LIN {X 0,Y 171.354,Z 701.949,A -85,B 0,C 180,E1 7628.432,E2 7628.432} C_VEL
LIN {X 0,Y 180.536,Z 691.15,A -85,B 0,C 180,E1 7622.276,E2 7622.276} C_VEL
LIN {X 0,Y 190.224,Z 679.335,A -85,B 0,C 180,E1 7617.222,E2 7617.222} C_VEL
LIN {X 0,Y 200.427,Z 666.059,A -85,B 0,C 180,E1 7612.87,E2 7612.87} C_VEL
LIN {X 0,Y 210.868,Z 651.279,A -85,B 0,C 180,E1 7609.131,E2 7609.131} C_VEL
LIN {X 0,Y 221.307,Z 634.876,A -85,B 0,C 180,E1 7605.912,E2 7605.912} C_VEL
LIN {X 0,Y 231.183,Z 617.293,A -85,B 0,C 180,E1 7603.218,E2 7603.218} C_VEL
LIN {X 0,Y 240.325,Z 598.504,A -85,B 0,C 180,E1 7600.964,E2 7600.964} C_VEL
LIN {X 0,Y 248.227,Z 579.366,A -85,B 0,C 180,E1 7599.16,E2 7599.16} C_VEL
LIN {X 0,Y 255.118,Z 559.071,A -85,B 0,C 180,E1 7597.658,E2 7597.658} C_VEL
LIN {X 0,Y 260.735,Z 538.067,A -85,B 0,C 180,E1 7596.463,E2 7596.463} C_VEL
LIN {X 0,Y 268.642,Z 500.013,A -85,B 0,C 180,E1 7594.871,E2 7594.871} C_VEL
LIN {X 0,Y 278.866,Z 448.019,A -85,B 0,C 180,E1 7593.295,E2 7593.295} C_VEL
LIN {X 0,Y 287.897,Z 394.54,A -85,B 0,C 180,E1 7591.964,E2 7591.964} C_VEL
LIN {X 0,Y 288.757,Z 388.485,A -85,B 0,C 180,E1 7591.797,E2 7591.797} C_VEL
LIN {X 0,Y 284.444,Z 383.003,A -85,B 0,C 180,E1 7588.674,E2 7588.674} C_VEL
LIN {X 0,Y 280.996,Z 379.022,A -85,B 0,C 180,E1 7585.729,E2 7585.729} C_VEL
LIN {X 0,Y 276.103,Z 374.241,A -85,B 0,C 180,E1 7580.344,E2 7580.344} C_VEL
LIN {X 0,Y 273.477,Z 373.45,A -85,B 0,C 180,E1 7576.133,E2 7576.133} C_VEL
LIN {X 0,Y 271.437,Z 376.229,A -85,B 0,C 180,E1 7569.97,E2 7569.97} C_VEL
LIN {X 0,Y 271.324,Z 379.346,A -85,B 0,C 180,E1 7566.56,E2 7566.56} C_VEL
LIN {X 0,Y 271.923,Z 384.024,A -85,B 0,C 180,E1 7563.057,E2 7563.057} C_VEL
LIN {X 0,Y 273.747,Z 392.011,A -85,B 0,C 180,E1 7558.64,E2 7558.64} C_VEL
LIN {X 0,Y 274.886,Z 396.29,A -85,B 0,C 180,E1 7556.725,E2 7556.725} C_VEL
LIN {X 0,Y 275.274,Z 398.796,A -85,B 0,C 180,E1 7555.994,E2 7555.994} C_VEL
LIN {X 0,Y 275.387,Z 403.134,A -85,B 0,C 180,E1 7555.297,E2 7555.297} C_VEL
LIN {X 0,Y 275.024,Z 410.299,A -85,B 0,C 180,E1 7554.636,E2 7554.636} C_VEL
LIN {X 0,Y 273.575,Z 426.263,A -85,B 0,C 180,E1 7553.562,E2 7553.562} C_VEL
LIN {X 0,Y 273.448,Z 428.423,A -85,B 0,C 180,E1 7553.346,E2 7553.346} C_VEL
LIN {X 0,Y 272.402,Z 456.029,A -85,B 0,C 180,E1 7550.133,E2 7550.133} C_VEL
LIN {X 0,Y 272.268,Z 480.855,A -85,B 0,C 180,E1 7546.766,E2 7546.766} C_VEL
LIN {X 0,Y 272.455,Z 492.691,A -85,B 0,C 180,E1 7545.052,E2 7545.052} C_VEL
LIN {X 0,Y 265.485,Z 519.701,A -85,B 0,C 180,E1 7544.247,E2 7544.247} C_VEL
LIN {X 0,Y 255.03,Z 554.502,A -85,B 0,C 180,E1 7542.869,E2 7542.869} C_VEL
LIN {X 0,Y 244.48,Z 585.093,A -85,B 0,C 180,E1 7541.222,E2 7541.222} C_VEL
LIN {X 0,Y 236.563,Z 605.451,A -85,B 0,C 180,E1 7539.768,E2 7539.768} C_VEL
LIN {X 0,Y 227.635,Z 624.889,A -85,B 0,C 180,E1 7537.94,E2 7537.94} C_VEL
LIN {X 0,Y 218.204,Z 642.726,A -85,B 0,C 180,E1 7535.763,E2 7535.763} C_VEL
LIN {X 0,Y 208.39,Z 659.271,A -85,B 0,C 180,E1 7533.18,E2 7533.18} C_VEL
LIN {X 0,Y 198.054,Z 675.047,A -85,B 0,C 180,E1 7530.015,E2 7530.015} C_VEL
LIN {X 0,Y 187.626,Z 689.669,A -85,B 0,C 180,E1 7526.234,E2 7526.234} C_VEL
LIN {X 0,Y 177.269,Z 703.298,A -85,B 0,C 180,E1 7521.628,E2 7521.628} C_VEL
LIN {X 0,Y 167.612,Z 715.397,A -85,B 0,C 180,E1 7516.203,E2 7516.203} C_VEL
LIN {X 0,Y 159.1,Z 726.025,A -85,B 0,C 180,E1 7509.867,E2 7509.867} C_VEL
LIN {X 0,Y 152.219,Z 735.127,A -85,B 0,C 180,E1 7502.589,E2 7502.589} C_VEL
LIN {X 0,Y 147.567,Z 742.333,A -85,B 0,C 180,E1 7494.782,E2 7494.782} C_VEL
LIN {X 0,Y 145.172,Z 747.597,A -85,B 0,C 180,E1 7486.798,E2 7486.798} C_VEL
LIN {X 0,Y 144.601,Z 751.03,A -85,B 0,C 180,E1 7479.15,E2 7479.15} C_VEL
LIN {X 0,Y 144.814,Z 752.641,A -85,B 0,C 180,E1 7473.166,E2 7473.166} C_VEL
LIN {X 0,Y 144.816,Z 753.275,A -85,B 0,C 180,E1 7468.021,E2 7468.021} C_VEL
LIN {X 0,Y 144.519,Z 753.042,A -85,B 0,C 180,E1 7462.046,E2 7462.046} C_VEL
LIN {X 0,Y 144.929,Z 751.416,A -85,B 0,C 180,E1 7453.98,E2 7453.98} C_VEL
LIN {X 0,Y 147.594,Z 747.947,A -85,B 0,C 180,E1 7445.164,E2 7445.164} C_VEL
LIN {X 0,Y 153.035,Z 742.69,A -85,B 0,C 180,E1 7436.713,E2 7436.713} C_VEL
LIN {X 0,Y 161.282,Z 735.568,A -85,B 0,C 180,E1 7428.917,E2 7428.917} C_VEL
LIN {X 0,Y 172.223,Z 726.333,A -85,B 0,C 180,E1 7421.884,E2 7421.884} C_VEL
LIN {X 0,Y 185.117,Z 715.226,A -85,B 0,C 180,E1 7415.885,E2 7415.885} C_VEL
LIN {X 0,Y 189.553,Z 711.162,A -85,B 0,C 180,E1 7414.101,E2 7414.101} C_VEL
LIN {X 0,Y 177.044,Z 711.814,A -85,B 0,C 180,E1 7408.687,E2 7408.687} C_VEL
LIN {X 0,Y 164.866,Z 711.841,A -85,B 0,C 180,E1 7400.222,E2 7400.222} C_VEL
LIN {X 0,Y 156.934,Z 710.739,A -85,B 0,C 180,E1 7385.85,E2 7385.85} C_VEL
LIN {X 0,Y 167.659,Z 708.493,A -85,B 0,C 180,E1 7362.65,E2 7362.65} C_VEL
LIN {X 0,Y 180.213,Z 707.275,A -85,B 0,C 180,E1 7354.299,E2 7354.299} C_VEL
LIN {X 0,Y 168.721,Z 715.346,A -85,B 0,C 180,E1 7347.935,E2 7347.935} C_VEL
LIN {X 0,Y 159.559,Z 721.376,A -85,B 0,C 180,E1 7340.991,E2 7340.991} C_VEL
LIN {X 0,Y 152.377,Z 725.891,A -85,B 0,C 180,E1 7333.034,E2 7333.034} C_VEL
LIN {X 0,Y 147.772,Z 728.661,A -85,B 0,C 180,E1 7324.637,E2 7324.637} C_VEL
LIN {X 0,Y 145.581,Z 729.803,A -85,B 0,C 180,E1 7316.515,E2 7316.515} C_VEL
LIN {X 0,Y 144.885,Z 729.625,A -85,B 0,C 180,E1 7309.345,E2 7309.345} C_VEL
LIN {X 0,Y 144.897,Z 728.45,A -85,B 0,C 180,E1 7302.353,E2 7302.353} C_VEL
LIN {X 0,Y 145.734,Z 726.021,A -85,B 0,C 180,E1 7294.723,E2 7294.723} C_VEL
LIN {X 0,Y 148.261,Z 721.791,A -85,B 0,C 180,E1 7286.491,E2 7286.491} C_VEL
LIN {X 0,Y 152.759,Z 715.974,A -85,B 0,C 180,E1 7278.676,E2 7278.676} C_VEL
LIN {X 0,Y 158.986,Z 708.791,A -85,B 0,C 180,E1 7271.673,E2 7271.673} C_VEL
LIN {X 0,Y 167.002,Z 699.89,A -85,B 0,C 180,E1 7265.223,E2 7265.223} C_VEL
LIN {X 0,Y 176.613,Z 689.064,A -85,B 0,C 180,E1 7259.369,E2 7259.369} C_VEL
LIN {X 0,Y 187.046,Z 676.723,A -85,B 0,C 180,E1 7254.363,E2 7254.363} C_VEL
LIN {X 0,Y 197.931,Z 662.854,A -85,B 0,C 180,E1 7250.093,E2 7250.093} C_VEL
LIN {X 0,Y 208.956,Z 647.38,A -85,B 0,C 180,E1 7246.446,E2 7246.446} C_VEL
LIN {X 0,Y 219.545,Z 630.725,A -85,B 0,C 180,E1 7243.415,E2 7243.415} C_VEL
LIN {X 0,Y 229.485,Z 612.921,A -85,B 0,C 180,E1 7240.893,E2 7240.893} C_VEL
LIN {X 0,Y 238.591,Z 593.934,A -85,B 0,C 180,E1 7238.789,E2 7238.789} C_VEL
LIN {X 0,Y 246.367,Z 574.632,A -85,B 0,C 180,E1 7237.111,E2 7237.111} C_VEL
LIN {X 0,Y 253.084,Z 554.191,A -85,B 0,C 180,E1 7235.721,E2 7235.721} C_VEL
LIN {X 0,Y 258.439,Z 533.188,A -85,B 0,C 180,E1 7234.629,E2 7234.629} C_VEL
LIN {X 0,Y 267.711,Z 489.4,A -85,B 0,C 180,E1 7232.935,E2 7232.935} C_VEL
LIN {X 0,Y 278.293,Z 435.561,A -85,B 0,C 180,E1 7231.428,E2 7231.428} C_VEL
LIN {X 0,Y 285.226,Z 394.061,A -85,B 0,C 180,E1 7230.419,E2 7230.419} C_VEL
LIN {X 0,Y 282.138,Z 390.149,A -85,B 0,C 180,E1 7228.018,E2 7228.018} C_VEL
LIN {X 0,Y 279.285,Z 386.715,A -85,B 0,C 180,E1 7225.443,E2 7225.443} C_VEL
LIN {X 0,Y 274.726,Z 382.112,A -85,B 0,C 180,E1 7220.228,E2 7220.228} C_VEL
LIN {X 0,Y 272.265,Z 381.361,A -85,B 0,C 180,E1 7216.207,E2 7216.207} C_VEL
LIN {X 0,Y 270.259,Z 384.053,A -85,B 0,C 180,E1 7210.23,E2 7210.23} C_VEL
LIN {X 0,Y 270.076,Z 387.081,A -85,B 0,C 180,E1 7206.911,E2 7206.911} C_VEL
LIN {X 0,Y 270.572,Z 391.825,A -85,B 0,C 180,E1 7203.39,E2 7203.39} C_VEL
LIN {X 0,Y 272.158,Z 399.486,A -85,B 0,C 180,E1 7199.159,E2 7199.159} C_VEL
LIN {X 0,Y 274.034,Z 407.176,A -85,B 0,C 180,E1 7195.921,E2 7195.921} C_VEL
LIN {X 0,Y 274.431,Z 409.099,A -85,B 0,C 180,E1 7195.299,E2 7195.299} C_VEL
LIN {X 0,Y 273.448,Z 428.423,A -85,B 0,C 180,E1 7193.346,E2 7193.346} C_VEL
LIN {X 0,Y 272.835,Z 435.664,A -85,B 0,C 180,E1 7192.766,E2 7192.766} C_VEL
LIN {X 0,Y 269.949,Z 455.079,A -85,B 0,C 180,E1 7191.849,E2 7191.849} C_VEL
LIN {X 0,Y 269.308,Z 462.105,A -85,B 0,C 180,E1 7191.184,E2 7191.184} C_VEL
LIN {X 0,Y 268.716,Z 487.169,A -85,B 0,C 180,E1 7187.674,E2 7187.674} C_VEL
LIN {X 0,Y 268.656,Z 494.996,A -85,B 0,C 180,E1 7186.554,E2 7186.554} C_VEL
LIN {X 0,Y 261.061,Z 523.455,A -85,B 0,C 180,E1 7185.692,E2 7185.692} C_VEL
LIN {X 0,Y 251.381,Z 554.96,A -85,B 0,C 180,E1 7184.477,E2 7184.477} C_VEL
LIN {X 0,Y 240.328,Z 586.648,A -85,B 0,C 180,E1 7182.82,E2 7182.82} C_VEL
LIN {X 0,Y 232.121,Z 606.804,A -85,B 0,C 180,E1 7181.377,E2 7181.377} C_VEL
LIN {X 0,Y 222.982,Z 625.913,A -85,B 0,C 180,E1 7179.58,E2 7179.58} C_VEL
LIN {X 0,Y 213.041,Z 644.023,A -85,B 0,C 180,E1 7177.367,E2 7177.367} C_VEL
LIN {X 0,Y 202.454,Z 661.114,A -85,B 0,C 180,E1 7174.659,E2 7174.659} C_VEL
LIN {X 0,Y 191.415,Z 677.098,A -85,B 0,C 180,E1 7171.347,E2 7171.347} C_VEL
LIN {X 0,Y 180.41,Z 691.618,A -85,B 0,C 180,E1 7167.395,E2 7167.395} C_VEL
LIN {X 0,Y 169.71,Z 704.845,A -85,B 0,C 180,E1 7162.641,E2 7162.641} C_VEL
LIN {X 0,Y 159.702,Z 716.716,A -85,B 0,C 180,E1 7156.968,E2 7156.968} C_VEL
LIN {X 0,Y 151.072,Z 726.931,A -85,B 0,C 180,E1 7150.436,E2 7150.436} C_VEL
LIN {X 0,Y 144.036,Z 735.711,A -85,B 0,C 180,E1 7142.782,E2 7142.782} C_VEL
LIN {X 0,Y 139.377,Z 742.546,A -85,B 0,C 180,E1 7134.587,E2 7134.587} C_VEL
LIN {X 0,Y 137.058,Z 747.585,A -85,B 0,C 180,E1 7126.093,E2 7126.093} C_VEL
LIN {X 0,Y 136.647,Z 750.774,A -85,B 0,C 180,E1 7117.991,E2 7117.991} C_VEL
LIN {X 0,Y 136.885,Z 752.225,A -85,B 0,C 180,E1 7111.674,E2 7111.674} C_VEL
LIN {X 0,Y 136.759,Z 752.604,A -85,B 0,C 180,E1 7106.227,E2 7106.227} C_VEL
LIN {X 0,Y 136.505,Z 752.171,A -85,B 0,C 180,E1 7099.448,E2 7099.448} C_VEL
LIN {X 0,Y 137.628,Z 750.098,A -85,B 0,C 180,E1 7090.476,E2 7090.476} C_VEL
LIN {X 0,Y 141.567,Z 746.099,A -85,B 0,C 180,E1 7081.136,E2 7081.136} C_VEL
LIN {X 0,Y 148.697,Z 740.161,A -85,B 0,C 180,E1 7072.272,E2 7072.272} C_VEL
LIN {X 0,Y 159.02,Z 732.136,A -85,B 0,C 180,E1 7064.209,E2 7064.209} C_VEL
LIN {X 0,Y 171.416,Z 722.422,A -85,B 0,C 180,E1 7057.506,E2 7057.506} C_VEL
LIN {X 0,Y 179.894,Z 715.408,A -85,B 0,C 180,E1 7053.869,E2 7053.869} C_VEL
LIN {X 0,Y 165.312,Z 715.757,A -85,B 0,C 180,E1 7046.587,E2 7046.587} C_VEL
LIN {X 0,Y 154.531,Z 715.3,A -85,B 0,C 180,E1 7036.926,E2 7036.926} C_VEL
LIN {X 0,Y 149.737,Z 714.176,A -85,B 0,C 180,E1 7024.979,E2 7024.979} C_VEL
LIN {X 0,Y 160.695,Z 711.869,A -85,B 0,C 180,E1 7001.873,E2 7001.873} C_VEL
LIN {X 0,Y 171.293,Z 710.841,A -85,B 0,C 180,E1 6994.53,E2 6994.53} C_VEL
LIN {X 0,Y 159.716,Z 718.272,A -85,B 0,C 180,E1 6987.85,E2 6987.85} C_VEL
LIN {X 0,Y 150.382,Z 723.839,A -85,B 0,C 180,E1 6980.334,E2 6980.334} C_VEL
LIN {X 0,Y 143.279,Z 727.812,A -85,B 0,C 180,E1 6971.693,E2 6971.693} C_VEL
LIN {X 0,Y 139.036,Z 730,A -85,B 0,C 180,E1 6962.641,E2 6962.641} C_VEL
LIN {X 0,Y 137.309,Z 730.53,A -85,B 0,C 180,E1 6954.46,E2 6954.46} C_VEL
LIN {X 0,Y 136.849,Z 729.926,A -85,B 0,C 180,E1 6946.833,E2 6946.833} C_VEL
LIN {X 0,Y 137.087,Z 728.42,A -85,B 0,C 180,E1 6939.658,E2 6939.658} C_VEL
LIN {X 0,Y 138.427,Z 725.493,A -85,B 0,C 180,E1 6931.656,E2 6931.656} C_VEL
LIN {X 0,Y 141.776,Z 720.799,A -85,B 0,C 180,E1 6923.115,E2 6923.115} C_VEL
LIN {X 0,Y 147.636,Z 714.09,A -85,B 0,C 180,E1 6914.686,E2 6914.686} C_VEL
LIN {X 0,Y 155.429,Z 705.841,A -85,B 0,C 180,E1 6907.296,E2 6907.296} C_VEL
LIN {X 0,Y 165.159,Z 695.6,A -85,B 0,C 180,E1 6900.636,E2 6900.636} C_VEL
LIN {X 0,Y 175.99,Z 683.736,A -85,B 0,C 180,E1 6894.984,E2 6894.984} C_VEL
LIN {X 0,Y 187.476,Z 670.238,A -85,B 0,C 180,E1 6890.209,E2 6890.209} C_VEL
LIN {X 0,Y 198.57,Z 655.944,A -85,B 0,C 180,E1 6886.383,E2 6886.383} C_VEL
LIN {X 0,Y 209.615,Z 640.112,A -85,B 0,C 180,E1 6883.13,E2 6883.13} C_VEL
LIN {X 0,Y 220.041,Z 623.212,A -85,B 0,C 180,E1 6880.438,E2 6880.438} C_VEL
LIN {X 0,Y 229.654,Z 605.283,A -85,B 0,C 180,E1 6878.201,E2 6878.201} C_VEL
LIN {X 0,Y 238.329,Z 586.285,A -85,B 0,C 180,E1 6876.342,E2 6876.342} C_VEL
LIN {X 0,Y 245.568,Z 567.229,A -85,B 0,C 180,E1 6874.872,E2 6874.872} C_VEL
LIN {X 0,Y 251.885,Z 546.585,A -85,B 0,C 180,E1 6873.633,E2 6873.633} C_VEL
LIN {X 0,Y 258.787,Z 517.082,A -85,B 0,C 180,E1 6872.31,E2 6872.31} C_VEL
LIN {X 0,Y 267.881,Z 474.899,A -85,B 0,C 180,E1 6870.894,E2 6870.894} C_VEL
LIN {X 0,Y 278.004,Z 422.549,A -85,B 0,C 180,E1 6869.551,E2 6869.551} C_VEL
LIN {X 0,Y 281.82,Z 399.7,A -85,B 0,C 180,E1 6869.01,E2 6869.01} C_VEL
LIN {X 0,Y 277.532,Z 394.401,A -85,B 0,C 180,E1 6865.159,E2 6865.159} C_VEL
LIN {X 0,Y 273.269,Z 389.97,A -85,B 0,C 180,E1 6860.118,E2 6860.118} C_VEL
LIN {X 0,Y 271.014,Z 389.266,A -85,B 0,C 180,E1 6856.284,E2 6856.284} C_VEL
LIN {X 0,Y 268.974,Z 392.056,A -85,B 0,C 180,E1 6850.279,E2 6850.279} C_VEL
LIN {X 0,Y 268.78,Z 394.936,A -85,B 0,C 180,E1 6847.16,E2 6847.16} C_VEL
LIN {X 0,Y 269.175,Z 399.61,A -85,B 0,C 180,E1 6843.728,E2 6843.728} C_VEL
LIN {X 0,Y 270.526,Z 406.946,A -85,B 0,C 180,E1 6839.683,E2 6839.683} C_VEL
LIN {X 0,Y 272.103,Z 414.302,A -85,B 0,C 180,E1 6836.577,E2 6836.577} C_VEL
LIN {X 0,Y 270.3,Z 442.419,A -85,B 0,C 180,E1 6833.589,E2 6833.589} C_VEL
LIN {X 0,Y 269.308,Z 462.105,A -85,B 0,C 180,E1 6831.184,E2 6831.184} C_VEL
LIN {X 0,Y 268.709,Z 469.106,A -85,B 0,C 180,E1 6830.479,E2 6830.479} C_VEL
LIN {X 0,Y 265.764,Z 488.052,A -85,B 0,C 180,E1 6829.195,E2 6829.195} C_VEL
LIN {X 0,Y 265.158,Z 494.824,A -85,B 0,C 180,E1 6828.404,E2 6828.404} C_VEL
LIN {X 0,Y 264.979,Z 497.272,A -85,B 0,C 180,E1 6828.09,E2 6828.09} C_VEL
LIN {X 0,Y 256.396,Z 528.682,A -85,B 0,C 180,E1 6827.139,E2 6827.139} C_VEL
LIN {X 0,Y 245.452,Z 562.722,A -85,B 0,C 180,E1 6825.812,E2 6825.812} C_VEL
LIN {X 0,Y 235.247,Z 590.673,A -85,B 0,C 180,E1 6824.297,E2 6824.297} C_VEL
LIN {X 0,Y 227.439,Z 608.962,A -85,B 0,C 180,E1 6822.972,E2 6822.972} C_VEL
LIN {X 0,Y 217.978,Z 628.013,A -85,B 0,C 180,E1 6821.177,E2 6821.177} C_VEL
LIN {X 0,Y 207.383,Z 646.391,A -85,B 0,C 180,E1 6818.895,E2 6818.895} C_VEL
LIN {X 0,Y 196.267,Z 663.341,A -85,B 0,C 180,E1 6816.126,E2 6816.126} C_VEL
LIN {X 0,Y 184.568,Z 679.376,A -85,B 0,C 180,E1 6812.677,E2 6812.677} C_VEL
LIN {X 0,Y 173.275,Z 693.522,A -85,B 0,C 180,E1 6808.65,E2 6808.65} C_VEL
LIN {X 0,Y 162.092,Z 706.598,A -85,B 0,C 180,E1 6803.69,E2 6803.69} C_VEL
LIN {X 0,Y 151.554,Z 718.304,A -85,B 0,C 180,E1 6797.637,E2 6797.637} C_VEL
LIN {X 0,Y 142.644,Z 728.178,A -85,B 0,C 180,E1 6790.683,E2 6790.683} C_VEL
LIN {X 0,Y 135.559,Z 736.567,A -85,B 0,C 180,E1 6782.576,E2 6782.576} C_VEL
LIN {X 0,Y 130.99,Z 743.072,A -85,B 0,C 180,E1 6773.862,E2 6773.862} C_VEL
LIN {X 0,Y 128.899,Z 747.786,A -85,B 0,C 180,E1 6764.831,E2 6764.831} C_VEL
LIN {X 0,Y 128.716,Z 750.513,A -85,B 0,C 180,E1 6756.691,E2 6756.691} C_VEL
LIN {X 0,Y 128.939,Z 751.655,A -85,B 0,C 180,E1 6750.444,E2 6750.444} C_VEL
LIN {X 0,Y 128.695,Z 751.92,A -85,B 0,C 180,E1 6744.65,E2 6744.65} C_VEL
LIN {X 0,Y 128.67,Z 751.118,A -85,B 0,C 180,E1 6736.244,E2 6736.244} C_VEL
LIN {X 0,Y 130.795,Z 748.594,A -85,B 0,C 180,E1 6726.536,E2 6726.536} C_VEL
LIN {X 0,Y 136.327,Z 744.053,A -85,B 0,C 180,E1 6716.627,E2 6716.627} C_VEL
LIN {X 0,Y 145.281,Z 737.569,A -85,B 0,C 180,E1 6707.587,E2 6707.587} C_VEL
LIN {X 0,Y 156.702,Z 729.392,A -85,B 0,C 180,E1 6700.032,E2 6700.032} C_VEL
LIN {X 0,Y 170.19,Z 719.296,A -85,B 0,C 180,E1 6693.621,E2 6693.621} C_VEL
LIN {X 0,Y 154.36,Z 719.231,A -85,B 0,C 180,E1 6684.49,E2 6684.49} C_VEL
LIN {X 0,Y 143.397,Z 718.1,A -85,B 0,C 180,E1 6670.038,E2 6670.038} C_VEL
LIN {X 0,Y 154.109,Z 715.004,A -85,B 0,C 180,E1 6640.676,E2 6640.676} C_VEL
LIN {X 0,Y 162.224,Z 714.235,A -85,B 0,C 180,E1 6634.733,E2 6634.733} C_VEL
LIN {X 0,Y 150.963,Z 720.78,A -85,B 0,C 180,E1 6627.971,E2 6627.971} C_VEL
LIN {X 0,Y 141.536,Z 725.832,A -85,B 0,C 180,E1 6619.993,E2 6619.993} C_VEL
LIN {X 0,Y 134.84,Z 729.141,A -85,B 0,C 180,E1 6611.297,E2 6611.297} C_VEL
LIN {X 0,Y 130.765,Z 730.897,A -85,B 0,C 180,E1 6601.844,E2 6601.844} C_VEL
LIN {X 0,Y 129.159,Z 731.134,A -85,B 0,C 180,E1 6592.892,E2 6592.892} C_VEL
LIN {X 0,Y 128.875,Z 730.299,A -85,B 0,C 180,E1 6585.296,E2 6585.296} C_VEL
LIN {X 0,Y 129.368,Z 728.333,A -85,B 0,C 180,E1 6577.104,E2 6577.104} C_VEL
LIN {X 0,Y 131.435,Z 724.876,A -85,B 0,C 180,E1 6568.257,E2 6568.257} C_VEL
LIN {X 0,Y 135.782,Z 719.681,A -85,B 0,C 180,E1 6559.392,E2 6559.392} C_VEL
LIN {X 0,Y 142.46,Z 712.772,A -85,B 0,C 180,E1 6551.165,E2 6551.165} C_VEL
LIN {X 0,Y 151.325,Z 704.001,A -85,B 0,C 180,E1 6543.725,E2 6543.725} C_VEL
LIN {X 0,Y 161.537,Z 693.741,A -85,B 0,C 180,E1 6537.419,E2 6537.419} C_VEL
LIN {X 0,Y 172.62,Z 682.015,A -85,B 0,C 180,E1 6532.123,E2 6532.123} C_VEL
LIN {X 0,Y 184.126,Z 668.837,A -85,B 0,C 180,E1 6527.674,E2 6527.674} C_VEL
LIN {X 0,Y 195.756,Z 654.155,A -85,B 0,C 180,E1 6523.931,E2 6523.931} C_VEL
LIN {X 0,Y 207.256,Z 637.837,A -85,B 0,C 180,E1 6520.764,E2 6520.764} C_VEL
LIN {X 0,Y 218.052,Z 620.358,A -85,B 0,C 180,E1 6518.15,E2 6518.15} C_VEL
LIN {X 0,Y 227.942,Z 601.777,A -85,B 0,C 180,E1 6515.994,E2 6515.994} C_VEL
LIN {X 0,Y 236.523,Z 582.728,A -85,B 0,C 180,E1 6514.265,E2 6514.265} C_VEL
LIN {X 0,Y 243.955,Z 562.676,A -85,B 0,C 180,E1 6512.839,E2 6512.839} C_VEL
LIN {X 0,Y 250.174,Z 541.384,A -85,B 0,C 180,E1 6511.676,E2 6511.676} C_VEL
LIN {X 0,Y 259.603,Z 500.631,A -85,B 0,C 180,E1 6510.042,E2 6510.042} C_VEL
LIN {X 0,Y 269.641,Z 454.025,A -85,B 0,C 180,E1 6508.722,E2 6508.722} C_VEL
LIN {X 0,Y 278.539,Z 405.648,A -85,B 0,C 180,E1 6507.586,E2 6507.586} C_VEL
LIN {X 0,Y 275.56,Z 401.887,A -85,B 0,C 180,E1 6504.663,E2 6504.663} C_VEL
LIN {X 0,Y 271.804,Z 397.826,A -85,B 0,C 180,E1 6500.006,E2 6500.006} C_VEL
LIN {X 0,Y 269.673,Z 397.154,A -85,B 0,C 180,E1 6496.367,E2 6496.367} C_VEL
LIN {X 0,Y 267.682,Z 399.855,A -85,B 0,C 180,E1 6490.547,E2 6490.547} C_VEL
LIN {X 0,Y 267.443,Z 402.648,A -85,B 0,C 180,E1 6487.519,E2 6487.519} C_VEL
LIN {X 0,Y 267.718,Z 407.375,A -85,B 0,C 180,E1 6484.07,E2 6484.07} C_VEL
LIN {X 0,Y 268.86,Z 414.392,A -85,B 0,C 180,E1 6480.214,E2 6480.214} C_VEL
LIN {X 0,Y 269.859,Z 420.094,A -85,B 0,C 180,E1 6477.798,E2 6477.798} C_VEL
LIN {X 0,Y 267.706,Z 446.388,A -85,B 0,C 180,E1 6474.965,E2 6474.965} C_VEL
LIN {X 0,Y 266.016,Z 471.924,A -85,B 0,C 180,E1 6471.748,E2 6471.748} C_VEL
LIN {X 0,Y 265.158,Z 494.824,A -85,B 0,C 180,E1 6468.404,E2 6468.404} C_VEL
LIN {X 0,Y 264.609,Z 498.077,A -85,B 0,C 180,E1 6468.164,E2 6468.164} C_VEL
LIN {X 0,Y 263.21,Z 502.217,A -85,B 0,C 180,E1 6468.258,E2 6468.258} C_VEL
LIN {X 0,Y 258.133,Z 513.262,A -85,B 0,C 180,E1 6469.155,E2 6469.155} C_VEL
LIN {X 0,Y 256.778,Z 517.033,A -85,B 0,C 180,E1 6469.182,E2 6469.182} C_VEL
LIN {X 0,Y 246.767,Z 549.705,A -85,B 0,C 180,E1 6468.075,E2 6468.075} C_VEL
LIN {X 0,Y 235.377,Z 582.079,A -85,B 0,C 180,E1 6466.598,E2 6466.598} C_VEL
LIN {X 0,Y 226.9,Z 602.616,A -85,B 0,C 180,E1 6465.295,E2 6465.295} C_VEL
LIN {X 0,Y 217.706,Z 621.428,A -85,B 0,C 180,E1 6463.713,E2 6463.713} C_VEL
LIN {X 0,Y 207.444,Z 639.576,A -85,B 0,C 180,E1 6461.716,E2 6461.716} C_VEL
LIN {X 0,Y 196.658,Z 656.347,A -85,B 0,C 180,E1 6459.309,E2 6459.309} C_VEL
LIN {X 0,Y 185.1,Z 672.382,A -85,B 0,C 180,E1 6456.289,E2 6456.289} C_VEL
LIN {X 0,Y 173.381,Z 687.06,A -85,B 0,C 180,E1 6452.633,E2 6452.633} C_VEL
LIN {X 0,Y 161.435,Z 700.69,A -85,B 0,C 180,E1 6448.05,E2 6448.05} C_VEL
LIN {X 0,Y 150.046,Z 712.887,A -85,B 0,C 180,E1 6442.464,E2 6442.464} C_VEL
LIN {X 0,Y 139.708,Z 723.626,A -85,B 0,C 180,E1 6435.698,E2 6435.698} C_VEL
LIN {X 0,Y 131.417,Z 732.411,A -85,B 0,C 180,E1 6428.044,E2 6428.044} C_VEL
LIN {X 0,Y 125.206,Z 739.756,A -85,B 0,C 180,E1 6419.151,E2 6419.151} C_VEL
LIN {X 0,Y 121.7,Z 745.246,A -85,B 0,C 180,E1 6409.684,E2 6409.684} C_VEL
LIN {X 0,Y 120.666,Z 748.836,A -85,B 0,C 180,E1 6400.503,E2 6400.503} C_VEL
LIN {X 0,Y 120.892,Z 750.527,A -85,B 0,C 180,E1 6393.318,E2 6393.318} C_VEL
LIN {X 0,Y 120.884,Z 751.184,A -85,B 0,C 180,E1 6387.629,E2 6387.629} C_VEL
LIN {X 0,Y 120.547,Z 751.088,A -85,B 0,C 180,E1 6380.45,E2 6380.45} C_VEL
LIN {X 0,Y 121.482,Z 749.628,A -85,B 0,C 180,E1 6370.778,E2 6370.778} C_VEL
LIN {X 0,Y 125.495,Z 746.319,A -85,B 0,C 180,E1 6360.397,E2 6360.397} C_VEL
LIN {X 0,Y 133.3,Z 741.012,A -85,B 0,C 180,E1 6350.388,E2 6350.388} C_VEL
LIN {X 0,Y 143.943,Z 734.076,A -85,B 0,C 180,E1 6341.99,E2 6341.99} C_VEL
LIN {X 0,Y 157.18,Z 725.207,A -85,B 0,C 180,E1 6334.854,E2 6334.854} C_VEL
LIN {X 0,Y 160.523,Z 722.807,A -85,B 0,C 180,E1 6333.334,E2 6333.334} C_VEL
LIN {X 0,Y 145.642,Z 722.467,A -85,B 0,C 180,E1 6323.893,E2 6323.893} C_VEL
LIN {X 0,Y 135.208,Z 720.885,A -85,B 0,C 180,E1 6306.367,E2 6306.367} C_VEL
LIN {X 0,Y 149.221,Z 717.769,A -85,B 0,C 180,E1 6277.96,E2 6277.96} C_VEL
LIN {X 0,Y 153.292,Z 717.333,A -85,B 0,C 180,E1 6275.046,E2 6275.046} C_VEL
LIN {X 0,Y 141.241,Z 723.643,A -85,B 0,C 180,E1 6267.397,E2 6267.397} C_VEL
LIN {X 0,Y 131.452,Z 728.258,A -85,B 0,C 180,E1 6258.196,E2 6258.196} C_VEL
LIN {X 0,Y 125.188,Z 730.881,A -85,B 0,C 180,E1 6248.488,E2 6248.488} C_VEL
LIN {X 0,Y 121.937,Z 731.86,A -85,B 0,C 180,E1 6238.399,E2 6238.399} C_VEL
LIN {X 0,Y 120.975,Z 731.553,A -85,B 0,C 180,E1 6229.809,E2 6229.809} C_VEL
LIN {X 0,Y 120.982,Z 730.257,A -85,B 0,C 180,E1 6221.925,E2 6221.925} C_VEL
LIN {X 0,Y 122.119,Z 727.691,A -85,B 0,C 180,E1 6212.817,E2 6212.817} C_VEL
LIN {X 0,Y 125.261,Z 723.628,A -85,B 0,C 180,E1 6203.584,E2 6203.584} C_VEL
LIN {X 0,Y 131.312,Z 717.409,A -85,B 0,C 180,E1 6194.091,E2 6194.091} C_VEL
LIN {X 0,Y 139.562,Z 709.661,A -85,B 0,C 180,E1 6185.899,E2 6185.899} C_VEL
LIN {X 0,Y 149.926,Z 699.969,A -85,B 0,C 180,E1 6178.656,E2 6178.656} C_VEL
LIN {X 0,Y 161.459,Z 688.696,A -85,B 0,C 180,E1 6172.636,E2 6172.636} C_VEL
LIN {X 0,Y 173.637,Z 675.844,A -85,B 0,C 180,E1 6167.645,E2 6167.645} C_VEL
LIN {X 0,Y 185.363,Z 662.258,A -85,B 0,C 180,E1 6163.714,E2 6163.714} C_VEL
LIN {X 0,Y 197.348,Z 646.732,A -85,B 0,C 180,E1 6160.315,E2 6160.315} C_VEL
LIN {X 0,Y 209.062,Z 629.495,A -85,B 0,C 180,E1 6157.448,E2 6157.448} C_VEL
LIN {X 0,Y 219.942,Z 610.979,A -85,B 0,C 180,E1 6155.087,E2 6155.087} C_VEL
LIN {X 0,Y 229.439,Z 591.945,A -85,B 0,C 180,E1 6153.207,E2 6153.207} C_VEL
LIN {X 0,Y 237.831,Z 571.656,A -85,B 0,C 180,E1 6151.645,E2 6151.645} C_VEL
LIN {X 0,Y 244.659,Z 551.112,A -85,B 0,C 180,E1 6150.424,E2 6150.424} C_VEL
LIN {X 0,Y 251.802,Z 523.021,A -85,B 0,C 180,E1 6149.167,E2 6149.167} C_VEL
LIN {X 0,Y 261.39,Z 481.732,A -85,B 0,C 180,E1 6147.787,E2 6147.787} C_VEL
LIN {X 0,Y 271.741,Z 431.737,A -85,B 0,C 180,E1 6146.562,E2 6146.562} C_VEL
LIN {X 0,Y 275.361,Z 411.62,A -85,B 0,C 180,E1 6146.097,E2 6146.097} C_VEL
LIN {X 0,Y 273.14,Z 408.943,A -85,B 0,C 180,E1 6143.746,E2 6143.746} C_VEL
LIN {X 0,Y 270.249,Z 405.666,A -85,B 0,C 180,E1 6139.901,E2 6139.901} C_VEL
LIN {X 0,Y 268.296,Z 405.036,A -85,B 0,C 180,E1 6136.454,E2 6136.454} C_VEL
LIN {X 0,Y 266.302,Z 407.634,A -85,B 0,C 180,E1 6130.821,E2 6130.821} C_VEL
LIN {X 0,Y 266.006,Z 410.335,A -85,B 0,C 180,E1 6127.886,E2 6127.886} C_VEL
LIN {X 0,Y 266.157,Z 415.111,A -85,B 0,C 180,E1 6124.418,E2 6124.418} C_VEL
LIN {X 0,Y 267.114,Z 421.92,A -85,B 0,C 180,E1 6120.698,E2 6120.698} C_VEL
LIN {X 0,Y 267.66,Z 425.756,A -85,B 0,C 180,E1 6119.064,E2 6119.064} C_VEL
LIN {X 0,Y 264.823,Z 454.145,A -85,B 0,C 180,E1 6115.914,E2 6115.914} C_VEL
LIN {X 0,Y 262.74,Z 480.368,A -85,B 0,C 180,E1 6112.484,E2 6112.484} C_VEL
LIN {X 0,Y 261.59,Z 499.478,A -85,B 0,C 180,E1 6109.672,E2 6109.672} C_VEL
LIN {X 0,Y 256.778,Z 517.033,A -85,B 0,C 180,E1 6109.182,E2 6109.182} C_VEL
LIN {X 0,Y 254.311,Z 524.379,A -85,B 0,C 180,E1 6109.196,E2 6109.196} C_VEL
LIN {X 0,Y 246.54,Z 542.774,A -85,B 0,C 180,E1 6109.865,E2 6109.865} C_VEL
LIN {X 0,Y 243.816,Z 550.01,A -85,B 0,C 180,E1 6109.811,E2 6109.811} C_VEL
LIN {X 0,Y 233.133,Z 580.237,A -85,B 0,C 180,E1 6108.517,E2 6108.517} C_VEL
LIN {X 0,Y 224.777,Z 600.351,A -85,B 0,C 180,E1 6107.324,E2 6107.324} C_VEL
LIN {X 0,Y 215.958,Z 618.332,A -85,B 0,C 180,E1 6105.92,E2 6105.92} C_VEL
LIN {X 0,Y 205.839,Z 636.126,A -85,B 0,C 180,E1 6104.107,E2 6104.107} C_VEL
LIN {X 0,Y 194.691,Z 653.269,A -85,B 0,C 180,E1 6101.821,E2 6101.821} C_VEL
LIN {X 0,Y 183.088,Z 669.096,A -85,B 0,C 180,E1 6099.041,E2 6099.041} C_VEL
LIN {X 0,Y 171.206,Z 683.678,A -85,B 0,C 180,E1 6095.65,E2 6095.65} C_VEL
LIN {X 0,Y 159.28,Z 697.026,A -85,B 0,C 180,E1 6091.5,E2 6091.5} C_VEL
LIN {X 0,Y 146.981,Z 709.789,A -85,B 0,C 180,E1 6086.09,E2 6086.09} C_VEL
LIN {X 0,Y 135.602,Z 720.933,A -85,B 0,C 180,E1 6079.417,E2 6079.417} C_VEL
LIN {X 0,Y 126.212,Z 730.077,A -85,B 0,C 180,E1 6071.716,E2 6071.716} C_VEL
LIN {X 0,Y 118.587,Z 738.106,A -85,B 0,C 180,E1 6062.084,E2 6062.084} C_VEL
LIN {X 0,Y 114.197,Z 743.984,A -85,B 0,C 180,E1 6051.866,E2 6051.866} C_VEL
LIN {X 0,Y 112.717,Z 747.868,A -85,B 0,C 180,E1 6041.771,E2 6041.771} C_VEL
LIN {X 0,Y 112.91,Z 749.789,A -85,B 0,C 180,E1 6033.553,E2 6033.553} C_VEL
LIN {X 0,Y 112.93,Z 750.443,A -85,B 0,C 180,E1 6027.97,E2 6027.97} C_VEL
LIN {X 0,Y 112.568,Z 750.488,A -85,B 0,C 180,E1 6020.369,E2 6020.369} C_VEL
LIN {X 0,Y 113.637,Z 749.148,A -85,B 0,C 180,E1 6009.93,E2 6009.93} C_VEL
LIN {X 0,Y 118.209,Z 745.904,A -85,B 0,C 180,E1 5998.68,E2 5998.68} C_VEL
LIN {X 0,Y 126.547,Z 740.832,A -85,B 0,C 180,E1 5988.417,E2 5988.417} C_VEL
LIN {X 0,Y 138.507,Z 733.698,A -85,B 0,C 180,E1 5979.428,E2 5979.428} C_VEL
LIN {X 0,Y 150.869,Z 726.021,A -85,B 0,C 180,E1 5973.03,E2 5973.03} C_VEL
LIN {X 0,Y 136.9,Z 725.437,A -85,B 0,C 180,E1 5963.227,E2 5963.227} C_VEL
LIN {X 0,Y 127.754,Z 723.806,A -85,B 0,C 180,E1 5946.289,E2 5946.289} C_VEL
LIN {X 0,Y 140.941,Z 720.674,A -85,B 0,C 180,E1 5917.913,E2 5917.913} C_VEL
LIN {X 0,Y 144.162,Z 720.373,A -85,B 0,C 180,E1 5915.311,E2 5915.311} C_VEL
LIN {X 0,Y 132.035,Z 726.048,A -85,B 0,C 180,E1 5907.202,E2 5907.202} C_VEL
LIN {X 0,Y 122.738,Z 729.901,A -85,B 0,C 180,E1 5897.845,E2 5897.845} C_VEL
LIN {X 0,Y 116.625,Z 732.049,A -85,B 0,C 180,E1 5887.497,E2 5887.497} C_VEL
LIN {X 0,Y 113.728,Z 732.566,A -85,B 0,C 180,E1 5877.205,E2 5877.205} C_VEL
LIN {X 0,Y 112.936,Z 731.902,A -85,B 0,C 180,E1 5868.052,E2 5868.052} C_VEL
LIN {X 0,Y 113.144,Z 730.434,A -85,B 0,C 180,E1 5859.667,E2 5859.667} C_VEL
LIN {X 0,Y 114.789,Z 727.516,A -85,B 0,C 180,E1 5850.001,E2 5850.001} C_VEL
LIN {X 0,Y 119.009,Z 722.831,A -85,B 0,C 180,E1 5839.839,E2 5839.839} C_VEL
LIN {X 0,Y 125.9,Z 716.472,A -85,B 0,C 180,E1 5830.516,E2 5830.516} C_VEL
LIN {X 0,Y 135.245,Z 708.308,A -85,B 0,C 180,E1 5822.242,E2 5822.242} C_VEL
LIN {X 0,Y 146.667,Z 698.143,A -85,B 0,C 180,E1 5815.066,E2 5815.066} C_VEL
LIN {X 0,Y 158.466,Z 686.99,A -85,B 0,C 180,E1 5809.467,E2 5809.467} C_VEL
LIN {X 0,Y 171.383,Z 673.681,A -85,B 0,C 180,E1 5804.623,E2 5804.623} C_VEL
LIN {X 0,Y 183.692,Z 659.588,A -85,B 0,C 180,E1 5800.836,E2 5800.836} C_VEL
LIN {X 0,Y 196.2,Z 643.463,A -85,B 0,C 180,E1 5797.586,E2 5797.586} C_VEL
LIN {X 0,Y 207.555,Z 626.742,A -85,B 0,C 180,E1 5795.021,E2 5795.021} C_VEL
LIN {X 0,Y 218.361,Z 608.293,A -85,B 0,C 180,E1 5792.836,E2 5792.836} C_VEL
LIN {X 0,Y 227.709,Z 589.447,A -85,B 0,C 180,E1 5791.104,E2 5791.104} C_VEL
LIN {X 0,Y 235.896,Z 569.492,A -85,B 0,C 180,E1 5789.669,E2 5789.669} C_VEL
LIN {X 0,Y 242.67,Z 548.804,A -85,B 0,C 180,E1 5788.522,E2 5788.522} C_VEL
LIN {X 0,Y 251.957,Z 512.333,A -85,B 0,C 180,E1 5787.034,E2 5787.034} C_VEL
LIN {X 0,Y 261.592,Z 471.098,A -85,B 0,C 180,E1 5785.826,E2 5785.826} C_VEL
LIN {X 0,Y 271.58,Z 422.04,A -85,B 0,C 180,E1 5784.715,E2 5784.715} C_VEL
LIN {X 0,Y 272.327,Z 417.667,A -85,B 0,C 180,E1 5784.572,E2 5784.572} C_VEL
LIN {X 0,Y 268.555,Z 413.462,A -85,B 0,C 180,E1 5779.619,E2 5779.619} C_VEL
LIN {X 0,Y 266.863,Z 412.907,A -85,B 0,C 180,E1 5776.545,E2 5776.545} C_VEL
LIN {X 0,Y 264.859,Z 415.458,A -85,B 0,C 180,E1 5771.035,E2 5771.035} C_VEL
LIN {X 0,Y 264.531,Z 418.012,A -85,B 0,C 180,E1 5768.259,E2 5768.259} C_VEL
LIN {X 0,Y 264.565,Z 422.834,A -85,B 0,C 180,E1 5764.77,E2 5764.77} C_VEL
LIN {X 0,Y 265.313,Z 429.426,A -85,B 0,C 180,E1 5761.188,E2 5761.188} C_VEL
LIN {X 0,Y 265.512,Z 431.556,A -85,B 0,C 180,E1 5760.324,E2 5760.324} C_VEL
LIN {X 0,Y 262.124,Z 460.31,A -85,B 0,C 180,E1 5757.063,E2 5757.063} C_VEL
LIN {X 0,Y 259.613,Z 486.376,A -85,B 0,C 180,E1 5753.563,E2 5753.563} C_VEL
LIN {X 0,Y 258.39,Z 501.571,A -85,B 0,C 180,E1 5751.29,E2 5751.29} C_VEL
LIN {X 0,Y 248.519,Z 535.696,A -85,B 0,C 180,E1 5750.298,E2 5750.298} C_VEL
LIN {X 0,Y 243.816,Z 550.01,A -85,B 0,C 180,E1 5749.811,E2 5749.811} C_VEL
LIN {X 0,Y 241.066,Z 557.266,A -85,B 0,C 180,E1 5749.767,E2 5749.767} C_VEL
LIN {X 0,Y 232.138,Z 576.405,A -85,B 0,C 180,E1 5750.386,E2 5750.386} C_VEL
LIN {X 0,Y 229.54,Z 582.459,A -85,B 0,C 180,E1 5750.271,E2 5750.271} C_VEL
LIN {X 0,Y 220.946,Z 602.34,A -85,B 0,C 180,E1 5749.112,E2 5749.112} C_VEL
LIN {X 0,Y 211.352,Z 621.037,A -85,B 0,C 180,E1 5747.661,E2 5747.661} C_VEL
LIN {X 0,Y 200.145,Z 639.801,A -85,B 0,C 180,E1 5745.733,E2 5745.733} C_VEL
LIN {X 0,Y 188.024,Z 657.303,A -85,B 0,C 180,E1 5743.313,E2 5743.313} C_VEL
LIN {X 0,Y 175.572,Z 673.18,A -85,B 0,C 180,E1 5740.368,E2 5740.368} C_VEL
LIN {X 0,Y 163.14,Z 687.411,A -85,B 0,C 180,E1 5736.827,E2 5736.827} C_VEL
LIN {X 0,Y 150.081,Z 700.987,A -85,B 0,C 180,E1 5732.204,E2 5732.204} C_VEL
LIN {X 0,Y 137.593,Z 713.015,A -85,B 0,C 180,E1 5726.478,E2 5726.478} C_VEL
LIN {X 0,Y 126.281,Z 723.41,A -85,B 0,C 180,E1 5719.472,E2 5719.472} C_VEL
LIN {X 0,Y 116.491,Z 732.374,A -85,B 0,C 180,E1 5710.716,E2 5710.716} C_VEL
LIN {X 0,Y 109.533,Z 739.383,A -85,B 0,C 180,E1 5700.742,E2 5700.742} C_VEL
LIN {X 0,Y 105.679,Z 744.588,A -85,B 0,C 180,E1 5689.913,E2 5689.913} C_VEL
LIN {X 0,Y 104.709,Z 747.927,A -85,B 0,C 180,E1 5679.341,E2 5679.341} C_VEL
LIN {X 0,Y 104.985,Z 749.307,A -85,B 0,C 180,E1 5672.182,E2 5672.182} C_VEL
LIN {X 0,Y 104.864,Z 749.842,A -85,B 0,C 180,E1 5666.172,E2 5666.172} C_VEL
LIN {X 0,Y 104.676,Z 749.599,A -85,B 0,C 180,E1 5656.746,E2 5656.746} C_VEL
LIN {X 0,Y 107.005,Z 747.809,A -85,B 0,C 180,E1 5645.005,E2 5645.005} C_VEL
LIN {X 0,Y 113.502,Z 744.099,A -85,B 0,C 180,E1 5633.199,E2 5633.199} C_VEL
LIN {X 0,Y 124.049,Z 738.458,A -85,B 0,C 180,E1 5622.82,E2 5622.82} C_VEL
LIN {X 0,Y 137.234,Z 731.213,A -85,B 0,C 180,E1 5614.582,E2 5614.582} C_VEL
LIN {X 0,Y 140.98,Z 728.956,A -85,B 0,C 180,E1 5612.615,E2 5612.615} C_VEL
LIN {X 0,Y 127.052,Z 728.036,A -85,B 0,C 180,E1 5601.222,E2 5601.222} C_VEL
LIN {X 0,Y 120.05,Z 725.9,A -85,B 0,C 180,E1 5579.998,E2 5579.998} C_VEL
LIN {X 0,Y 135.017,Z 723.116,A -85,B 0,C 180,E1 5555.627,E2 5555.627} C_VEL
LIN {X 0,Y 122.73,Z 728.218,A -85,B 0,C 180,E1 5546.916,E2 5546.916} C_VEL
LIN {X 0,Y 113.335,Z 731.552,A -85,B 0,C 180,E1 5536.516,E2 5536.516} C_VEL
LIN {X 0,Y 107.641,Z 733.086,A -85,B 0,C 180,E1 5525.164,E2 5525.164} C_VEL
LIN {X 0,Y 105.354,Z 733.073,A -85,B 0,C 180,E1 5514.34,E2 5514.34} C_VEL
LIN {X 0,Y 104.95,Z 732.101,A -85,B 0,C 180,E1 5504.907,E2 5504.907} C_VEL
LIN {X 0,Y 105.626,Z 730.058,A -85,B 0,C 180,E1 5495.433,E2 5495.433} C_VEL
LIN {X 0,Y 108.476,Z 726.45,A -85,B 0,C 180,E1 5484.712,E2 5484.712} C_VEL
LIN {X 0,Y 114.278,Z 721.083,A -85,B 0,C 180,E1 5474.25,E2 5474.25} C_VEL
LIN {X 0,Y 122.822,Z 714.001,A -85,B 0,C 180,E1 5464.957,E2 5464.957} C_VEL
LIN {X 0,Y 133.744,Z 705.026,A -85,B 0,C 180,E1 5456.925,E2 5456.925} C_VEL
LIN {X 0,Y 145.918,Z 694.531,A -85,B 0,C 180,E1 5450.413,E2 5450.413} C_VEL
LIN {X 0,Y 158.768,Z 682.534,A -85,B 0,C 180,E1 5445.144,E2 5445.144} C_VEL
LIN {X 0,Y 171.844,Z 669.033,A -85,B 0,C 180,E1 5440.853,E2 5440.853} C_VEL
LIN {X 0,Y 184.826,Z 653.976,A -85,B 0,C 180,E1 5437.324,E2 5437.324} C_VEL
LIN {X 0,Y 197.495,Z 637.24,A -85,B 0,C 180,E1 5434.39,E2 5434.39} C_VEL
LIN {X 0,Y 209.279,Z 619.248,A -85,B 0,C 180,E1 5432.002,E2 5432.002} C_VEL
LIN {X 0,Y 219.609,Z 600.737,A -85,B 0,C 180,E1 5430.112,E2 5430.112} C_VEL
LIN {X 0,Y 228.799,Z 581.075,A -85,B 0,C 180,E1 5428.554,E2 5428.554} C_VEL
LIN {X 0,Y 236.345,Z 561.235,A -85,B 0,C 180,E1 5427.327,E2 5427.327} C_VEL
LIN {X 0,Y 242.78,Z 539.592,A -85,B 0,C 180,E1 5426.299,E2 5426.299} C_VEL
LIN {X 0,Y 253.369,Z 497.658,A -85,B 0,C 180,E1 5424.802,E2 5424.802} C_VEL
LIN {X 0,Y 263.805,Z 452.056,A -85,B 0,C 180,E1 5423.688,E2 5423.688} C_VEL
LIN {X 0,Y 269.328,Z 424.177,A -85,B 0,C 180,E1 5423.059,E2 5423.059} C_VEL
LIN {X 0,Y 266.898,Z 421.277,A -85,B 0,C 180,E1 5419.477,E2 5419.477} C_VEL
LIN {X 0,Y 265.361,Z 420.762,A -85,B 0,C 180,E1 5416.641,E2 5416.641} C_VEL
LIN {X 0,Y 263.412,Z 423.16,A -85,B 0,C 180,E1 5411.385,E2 5411.385} C_VEL
LIN {X 0,Y 263,Z 425.804,A -85,B 0,C 180,E1 5408.527,E2 5408.527} C_VEL
LIN {X 0,Y 262.942,Z 430.943,A -85,B 0,C 180,E1 5404.866,E2 5404.866} C_VEL
LIN {X 0,Y 263.473,Z 437.112,A -85,B 0,C 180,E1 5401.618,E2 5401.618} C_VEL
LIN {X 0,Y 259.734,Z 464.876,A -85,B 0,C 180,E1 5398.429,E2 5398.429} C_VEL
LIN {X 0,Y 256.603,Z 491.212,A -85,B 0,C 180,E1 5394.831,E2 5394.831} C_VEL
LIN {X 0,Y 255.344,Z 503.861,A -85,B 0,C 180,E1 5392.942,E2 5392.942} C_VEL
LIN {X 0,Y 245.354,Z 537.684,A -85,B 0,C 180,E1 5391.998,E2 5391.998} C_VEL
LIN {X 0,Y 234.438,Z 569.46,A -85,B 0,C 180,E1 5390.867,E2 5390.867} C_VEL
LIN {X 0,Y 229.54,Z 582.459,A -85,B 0,C 180,E1 5390.271,E2 5390.271} C_VEL
LIN {X 0,Y 226.345,Z 589.548,A -85,B 0,C 180,E1 5390.141,E2 5390.141} C_VEL
LIN {X 0,Y 216.403,Z 606.955,A -85,B 0,C 180,E1 5390.539,E2 5390.539} C_VEL
LIN {X 0,Y 212.573,Z 613.631,A -85,B 0,C 180,E1 5390.3,E2 5390.3} C_VEL
LIN {X 0,Y 201.897,Z 632.038,A -85,B 0,C 180,E1 5388.682,E2 5388.682} C_VEL
LIN {X 0,Y 190.044,Z 649.684,A -85,B 0,C 180,E1 5386.616,E2 5386.616} C_VEL
LIN {X 0,Y 176.899,Z 666.786,A -85,B 0,C 180,E1 5383.916,E2 5383.916} C_VEL
LIN {X 0,Y 164.142,Z 681.491,A -85,B 0,C 180,E1 5380.763,E2 5380.763} C_VEL
LIN {X 0,Y 150.387,Z 695.747,A -85,B 0,C 180,E1 5376.563,E2 5376.563} C_VEL
LIN {X 0,Y 136.85,Z 708.449,A -85,B 0,C 180,E1 5371.252,E2 5371.252} C_VEL
LIN {X 0,Y 124.054,Z 719.6,A -85,B 0,C 180,E1 5364.492,E2 5364.492} C_VEL
LIN {X 0,Y 112.714,Z 729.194,A -85,B 0,C 180,E1 5355.932,E2 5355.932} C_VEL
LIN {X 0,Y 104.138,Z 736.81,A -85,B 0,C 180,E1 5345.85,E2 5345.85} C_VEL
LIN {X 0,Y 98.73,Z 742.673,A -85,B 0,C 180,E1 5334.298,E2 5334.298} C_VEL
LIN {X 0,Y 96.809,Z 746.407,A -85,B 0,C 180,E1 5323.132,E2 5323.132} C_VEL
LIN {X 0,Y 96.961,Z 748.398,A -85,B 0,C 180,E1 5313.546,E2 5313.546} C_VEL
LIN {X 0,Y 96.97,Z 749.032,A -85,B 0,C 180,E1 5307.635,E2 5307.635} C_VEL
LIN {X 0,Y 96.618,Z 749.15,A -85,B 0,C 180,E1 5299.264,E2 5299.264} C_VEL
LIN {X 0,Y 98.194,Z 747.992,A -85,B 0,C 180,E1 5287.235,E2 5287.235} C_VEL
LIN {X 0,Y 103.875,Z 745.077,A -85,B 0,C 180,E1 5274.721,E2 5274.721} C_VEL
LIN {X 0,Y 114.095,Z 740.197,A -85,B 0,C 180,E1 5263.333,E2 5263.333} C_VEL
LIN {X 0,Y 127.912,Z 733.354,A -85,B 0,C 180,E1 5254.045,E2 5254.045} C_VEL
LIN {X 0,Y 131.245,Z 731.573,A -85,B 0,C 180,E1 5252.225,E2 5252.225} C_VEL
LIN {X 0,Y 117.701,Z 730.358,A -85,B 0,C 180,E1 5239.346,E2 5239.346} C_VEL
LIN {X 0,Y 112.65,Z 728.218,A -85,B 0,C 180,E1 5218.472,E2 5218.472} C_VEL
LIN {X 0,Y 125.866,Z 725.693,A -85,B 0,C 180,E1 5196.002,E2 5196.002} C_VEL
LIN {X 0,Y 113.565,Z 730.155,A -85,B 0,C 180,E1 5186.764,E2 5186.764} C_VEL
LIN {X 0,Y 104.336,Z 732.894,A -85,B 0,C 180,E1 5175.606,E2 5175.606} C_VEL
LIN {X 0,Y 99.109,Z 733.912,A -85,B 0,C 180,E1 5163.703,E2 5163.703} C_VEL
LIN {X 0,Y 97.234,Z 733.61,A -85,B 0,C 180,E1 5153.003,E2 5153.003} C_VEL
LIN {X 0,Y 97.012,Z 732.37,A -85,B 0,C 180,E1 5143.106,E2 5143.106} C_VEL
LIN {X 0,Y 98.162,Z 730.052,A -85,B 0,C 180,E1 5132.336,E2 5132.336} C_VEL
LIN {X 0,Y 101.93,Z 726.085,A -85,B 0,C 180,E1 5120.971,E2 5120.971} C_VEL
LIN {X 0,Y 108.917,Z 720.34,A -85,B 0,C 180,E1 5110.145,E2 5110.145} C_VEL
LIN {X 0,Y 118.724,Z 712.84,A -85,B 0,C 180,E1 5100.761,E2 5100.761} C_VEL
LIN {X 0,Y 130.206,Z 703.907,A -85,B 0,C 180,E1 5093.205,E2 5093.205} C_VEL
LIN {X 0,Y 143.327,Z 693.026,A -85,B 0,C 180,E1 5086.871,E2 5086.871} C_VEL
LIN {X 0,Y 156.952,Z 680.608,A -85,B 0,C 180,E1 5081.812,E2 5081.812} C_VEL
LIN {X 0,Y 170.678,Z 666.63,A -85,B 0,C 180,E1 5077.735,E2 5077.735} C_VEL
LIN {X 0,Y 184.191,Z 650.973,A -85,B 0,C 180,E1 5074.401,E2 5074.401} C_VEL
LIN {X 0,Y 196.476,Z 634.694,A -85,B 0,C 180,E1 5071.805,E2 5071.805} C_VEL
LIN {X 0,Y 207.758,Z 617.397,A -85,B 0,C 180,E1 5069.695,E2 5069.695} C_VEL
LIN {X 0,Y 217.92,Z 599.141,A -85,B 0,C 180,E1 5067.966,E2 5067.966} C_VEL
LIN {X 0,Y 226.456,Z 580.951,A -85,B 0,C 180,E1 5066.609,E2 5066.609} C_VEL
LIN {X 0,Y 233.734,Z 562.172,A -85,B 0,C 180,E1 5065.497,E2 5065.497} C_VEL
LIN {X 0,Y 240.173,Z 541.13,A -85,B 0,C 180,E1 5064.528,E2 5064.528} C_VEL
LIN {X 0,Y 250.642,Z 501.065,A -85,B 0,C 180,E1 5063.128,E2 5063.128} C_VEL
LIN {X 0,Y 260.832,Z 458.271,A -85,B 0,C 180,E1 5062.109,E2 5062.109} C_VEL
LIN {X 0,Y 266.504,Z 430.781,A -85,B 0,C 180,E1 5061.515,E2 5061.515} C_VEL
LIN {X 0,Y 265.207,Z 429.089,A -85,B 0,C 180,E1 5059.377,E2 5059.377} C_VEL
LIN {X 0,Y 263.697,Z 428.695,A -85,B 0,C 180,E1 5056.522,E2 5056.522} C_VEL
LIN {X 0,Y 261.785,Z 431.078,A -85,B 0,C 180,E1 5051.456,E2 5051.456} C_VEL
LIN {X 0,Y 261.377,Z 433.571,A -85,B 0,C 180,E1 5048.802,E2 5048.802} C_VEL
LIN {X 0,Y 261.173,Z 438.576,A -85,B 0,C 180,E1 5045.273,E2 5045.273} C_VEL
LIN {X 0,Y 261.372,Z 443.098,A -85,B 0,C 180,E1 5042.879,E2 5042.879} C_VEL
LIN {X 0,Y 257.314,Z 470.03,A -85,B 0,C 180,E1 5039.736,E2 5039.736} C_VEL
LIN {X 0,Y 253.659,Z 496.48,A -85,B 0,C 180,E1 5036.065,E2 5036.065} C_VEL
LIN {X 0,Y 252.482,Z 506.171,A -85,B 0,C 180,E1 5034.626,E2 5034.626} C_VEL
LIN {X 0,Y 241.201,Z 543.195,A -85,B 0,C 180,E1 5033.638,E2 5033.638} C_VEL
LIN {X 0,Y 229.455,Z 576.426,A -85,B 0,C 180,E1 5032.454,E2 5032.454} C_VEL
LIN {X 0,Y 221.093,Z 596.422,A -85,B 0,C 180,E1 5031.446,E2 5031.446} C_VEL
LIN {X 0,Y 212.573,Z 613.631,A -85,B 0,C 180,E1 5030.3,E2 5030.3} C_VEL
LIN {X 0,Y 208.55,Z 620.33,A -85,B 0,C 180,E1 5030.021,E2 5030.021} C_VEL
LIN {X 0,Y 196.562,Z 636.416,A -85,B 0,C 180,E1 5030.124,E2 5030.124} C_VEL
LIN {X 0,Y 192.022,Z 642.509,A -85,B 0,C 180,E1 5029.732,E2 5029.732} C_VEL
LIN {X 0,Y 179.701,Z 659.051,A -85,B 0,C 180,E1 5027.548,E2 5027.548} C_VEL
LIN {X 0,Y 166.35,Z 674.805,A -85,B 0,C 180,E1 5024.729,E2 5024.729} C_VEL
LIN {X 0,Y 152.208,Z 689.522,A -85,B 0,C 180,E1 5021.073,E2 5021.073} C_VEL
LIN {X 0,Y 138.407,Z 702.387,A -85,B 0,C 180,E1 5016.555,E2 5016.555} C_VEL
LIN {X 0,Y 124.909,Z 713.893,A -85,B 0,C 180,E1 5010.751,E2 5010.751} C_VEL
LIN {X 0,Y 112.298,Z 723.985,A -85,B 0,C 180,E1 5003.256,E2 5003.256} C_VEL
LIN {X 0,Y 101.419,Z 732.577,A -85,B 0,C 180,E1 4993.638,E2 4993.638} C_VEL
LIN {X 0,Y 93.667,Z 739.26,A -85,B 0,C 180,E1 4982.257,E2 4982.257} C_VEL
LIN {X 0,Y 89.535,Z 744.139,A -85,B 0,C 180,E1 4969.572,E2 4969.572} C_VEL
LIN {X 0,Y 88.789,Z 747.019,A -85,B 0,C 180,E1 4957.721,E2 4957.721} C_VEL
LIN {X 0,Y 89.096,Z 748.153,A -85,B 0,C 180,E1 4949.999,E2 4949.999} C_VEL
LIN {X 0,Y 88.695,Z 748.524,A -85,B 0,C 180,E1 4942.224,E2 4942.224} C_VEL
LIN {X 0,Y 89.553,Z 747.94,A -85,B 0,C 180,E1 4929.69,E2 4929.69} C_VEL
LIN {X 0,Y 94.635,Z 745.646,A -85,B 0,C 180,E1 4915.945,E2 4915.945} C_VEL
LIN {X 0,Y 104.673,Z 741.388,A -85,B 0,C 180,E1 4903.449,E2 4903.449} C_VEL
LIN {X 0,Y 118.603,Z 735.246,A -85,B 0,C 180,E1 4893.424,E2 4893.424} C_VEL
LIN {X 0,Y 121.503,Z 733.879,A -85,B 0,C 180,E1 4891.778,E2 4891.778} C_VEL
LIN {X 0,Y 107.138,Z 732.157,A -85,B 0,C 180,E1 4874.593,E2 4874.593} C_VEL
LIN {X 0,Y 116.709,Z 728.112,A -85,B 0,C 180,E1 4836.448,E2 4836.448} C_VEL
LIN {X 0,Y 103.77,Z 732.111,A -85,B 0,C 180,E1 4825.961,E2 4825.961} C_VEL
LIN {X 0,Y 95.04,Z 734.174,A -85,B 0,C 180,E1 4813.977,E2 4813.977} C_VEL
LIN {X 0,Y 90.308,Z 734.618,A -85,B 0,C 180,E1 4800.618,E2 4800.618} C_VEL
LIN {X 0,Y 89.036,Z 733.815,A -85,B 0,C 180,E1 4789.379,E2 4789.379} C_VEL
LIN {X 0,Y 89.244,Z 732.327,A -85,B 0,C 180,E1 4779.025,E2 4779.025} C_VEL
LIN {X 0,Y 91.48,Z 729.331,A -85,B 0,C 180,E1 4766.868,E2 4766.868} C_VEL
LIN {X 0,Y 97.16,Z 724.562,A -85,B 0,C 180,E1 4754.482,E2 4754.482} C_VEL
LIN {X 0,Y 106.074,Z 718.11,A -85,B 0,C 180,E1 4743.704,E2 4743.704} C_VEL
LIN {X 0,Y 117.669,Z 709.837,A -85,B 0,C 180,E1 4734.704,E2 4734.704} C_VEL
LIN {X 0,Y 130.625,Z 700.081,A -85,B 0,C 180,E1 4727.656,E2 4727.656} C_VEL
LIN {X 0,Y 144.241,Z 688.884,A -85,B 0,C 180,E1 4722.123,E2 4722.123} C_VEL
LIN {X 0,Y 158.019,Z 676.279,A -85,B 0,C 180,E1 4717.728,E2 4717.728} C_VEL
LIN {X 0,Y 171.634,Z 662.225,A -85,B 0,C 180,E1 4714.186,E2 4714.186} C_VEL
LIN {X 0,Y 184.869,Z 646.675,A -85,B 0,C 180,E1 4711.292,E2 4711.292} C_VEL
LIN {X 0,Y 197.139,Z 630.115,A -85,B 0,C 180,E1 4708.968,E2 4708.968} C_VEL
LIN {X 0,Y 208.737,Z 611.877,A -85,B 0,C 180,E1 4707.008,E2 4707.008} C_VEL
LIN {X 0,Y 218.718,Z 593.24,A -85,B 0,C 180,E1 4705.464,E2 4705.464} C_VEL
LIN {X 0,Y 227.436,Z 573.564,A -85,B 0,C 180,E1 4704.187,E2 4704.187} C_VEL
LIN {X 0,Y 234.427,Z 554.085,A -85,B 0,C 180,E1 4703.201,E2 4703.201} C_VEL
LIN {X 0,Y 244.5,Z 518.366,A -85,B 0,C 180,E1 4701.85,E2 4701.85} C_VEL
LIN {X 0,Y 253.994,Z 481.248,A -85,B 0,C 180,E1 4700.844,E2 4700.844} C_VEL
LIN {X 0,Y 263.869,Z 437.373,A -85,B 0,C 180,E1 4699.973,E2 4699.973} C_VEL
LIN {X 0,Y 262.75,Z 436.567,A -85,B 0,C 180,E1 4697.948,E2 4697.948} C_VEL
LIN {X 0,Y 261.96,Z 436.608,A -85,B 0,C 180,E1 4696.407,E2 4696.407} C_VEL
LIN {X 0,Y 260.189,Z 438.802,A -85,B 0,C 180,E1 4691.752,E2 4691.752} C_VEL
LIN {X 0,Y 259.698,Z 441.45,A -85,B 0,C 180,E1 4688.971,E2 4688.971} C_VEL
LIN {X 0,Y 259.375,Z 446.482,A -85,B 0,C 180,E1 4685.531,E2 4685.531} C_VEL
LIN {X 0,Y 259.376,Z 449.097,A -85,B 0,C 180,E1 4684.159,E2 4684.159} C_VEL
LIN {X 0,Y 254.67,Z 477.323,A -85,B 0,C 180,E1 4680.788,E2 4680.788} C_VEL
LIN {X 0,Y 250.522,Z 503.854,A -85,B 0,C 180,E1 4677.011,E2 4677.011} C_VEL
LIN {X 0,Y 249.755,Z 508.497,A -85,B 0,C 180,E1 4676.339,E2 4676.339} C_VEL
LIN {X 0,Y 239.451,Z 542.052,A -85,B 0,C 180,E1 4675.508,E2 4675.508} C_VEL
LIN {X 0,Y 228.013,Z 574.439,A -85,B 0,C 180,E1 4674.465,E2 4674.465} C_VEL
LIN {X 0,Y 219.37,Z 594.963,A -85,B 0,C 180,E1 4673.519,E2 4673.519} C_VEL
LIN {X 0,Y 209.68,Z 614.101,A -85,B 0,C 180,E1 4672.32,E2 4672.32} C_VEL
LIN {X 0,Y 198.551,Z 632.763,A -85,B 0,C 180,E1 4670.753,E2 4670.753} C_VEL
LIN {X 0,Y 192.022,Z 642.509,A -85,B 0,C 180,E1 4669.732,E2 4669.732} C_VEL
LIN {X 0,Y 187.364,Z 648.561,A -85,B 0,C 180,E1 4669.293,E2 4669.293} C_VEL
LIN {X 0,Y 173.566,Z 663.185,A -85,B 0,C 180,E1 4669.003,E2 4669.003} C_VEL
LIN {X 0,Y 168.365,Z 668.643,A -85,B 0,C 180,E1 4668.388,E2 4668.388} C_VEL
LIN {X 0,Y 154.063,Z 683.723,A -85,B 0,C 180,E1 4665.237,E2 4665.237} C_VEL
LIN {X 0,Y 139.396,Z 697.445,A -85,B 0,C 180,E1 4661.171,E2 4661.171} C_VEL
LIN {X 0,Y 124.781,Z 709.7,A -85,B 0,C 180,E1 4655.881,E2 4655.881} C_VEL
LIN {X 0,Y 110.867,Z 720.396,A -85,B 0,C 180,E1 4648.954,E2 4648.954} C_VEL
LIN {X 0,Y 98.263,Z 729.58,A -85,B 0,C 180,E1 4639.741,E2 4639.741} C_VEL
LIN {X 0,Y 88.621,Z 736.783,A -85,B 0,C 180,E1 4628.354,E2 4628.354} C_VEL
LIN {X 0,Y 82.654,Z 742.224,A -85,B 0,C 180,E1 4614.874,E2 4614.874} C_VEL
LIN {X 0,Y 80.787,Z 745.69,A -85,B 0,C 180,E1 4601.42,E2 4601.42} C_VEL
LIN {X 0,Y 81.072,Z 747.163,A -85,B 0,C 180,E1 4592.119,E2 4592.119} C_VEL
LIN {X 0,Y 80.92,Z 747.677,A -85,B 0,C 180,E1 4585.747,E2 4585.747} C_VEL
LIN {X 0,Y 80.973,Z 747.689,A -85,B 0,C 180,E1 4573.499,E2 4573.499} C_VEL
LIN {X 0,Y 84.831,Z 746.189,A -85,B 0,C 180,E1 4558.76,E2 4558.76} C_VEL
LIN {X 0,Y 94.203,Z 742.749,A -85,B 0,C 180,E1 4544.672,E2 4544.672} C_VEL
LIN {X 0,Y 107.946,Z 737.452,A -85,B 0,C 180,E1 4533.525,E2 4533.525} C_VEL
LIN {X 0,Y 111.75,Z 735.902,A -85,B 0,C 180,E1 4531.259,E2 4531.259} C_VEL
LIN {X 0,Y 97.354,Z 733.482,A -85,B 0,C 180,E1 4507.671,E2 4507.671} C_VEL
LIN {X 0,Y 107.538,Z 730.263,A -85,B 0,C 180,E1 4476.998,E2 4476.998} C_VEL
LIN {X 0,Y 94.817,Z 733.569,A -85,B 0,C 180,E1 4466.018,E2 4466.018} C_VEL
LIN {X 0,Y 86.248,Z 735.107,A -85,B 0,C 180,E1 4453.081,E2 4453.081} C_VEL
LIN {X 0,Y 82.007,Z 735.135,A -85,B 0,C 180,E1 4439.191,E2 4439.191} C_VEL
LIN {X 0,Y 81.009,Z 734.184,A -85,B 0,C 180,E1 4427.232,E2 4427.232} C_VEL
LIN {X 0,Y 81.59,Z 732.329,A -85,B 0,C 180,E1 4415.627,E2 4415.627} C_VEL
LIN {X 0,Y 84.786,Z 729.08,A -85,B 0,C 180,E1 4402.548,E2 4402.548} C_VEL
LIN {X 0,Y 91.46,Z 724.252,A -85,B 0,C 180,E1 4390.191,E2 4390.191} C_VEL
LIN {X 0,Y 101.707,Z 717.485,A -85,B 0,C 180,E1 4379.257,E2 4379.257} C_VEL
LIN {X 0,Y 114.539,Z 708.852,A -85,B 0,C 180,E1 4370.414,E2 4370.414} C_VEL
LIN {X 0,Y 128.508,Z 698.71,A -85,B 0,C 180,E1 4363.649,E2 4363.649} C_VEL
LIN {X 0,Y 142.95,Z 687.08,A -85,B 0,C 180,E1 4358.43,E2 4358.43} C_VEL
LIN {X 0,Y 157.387,Z 673.986,A -85,B 0,C 180,E1 4354.324,E2 4354.324} C_VEL
LIN {X 0,Y 170.698,Z 660.334,A -85,B 0,C 180,E1 4351.22,E2 4351.22} C_VEL
LIN {X 0,Y 183.919,Z 644.839,A -85,B 0,C 180,E1 4348.601,E2 4348.601} C_VEL
LIN {X 0,Y 195.639,Z 629.084,A -85,B 0,C 180,E1 4346.572,E2 4346.572} C_VEL
LIN {X 0,Y 206.619,Z 611.965,A -85,B 0,C 180,E1 4344.861,E2 4344.861} C_VEL
LIN {X 0,Y 216.361,Z 594.123,A -85,B 0,C 180,E1 4343.464,E2 4343.464} C_VEL
LIN {X 0,Y 224.805,Z 575.638,A -85,B 0,C 180,E1 4342.315,E2 4342.315} C_VEL
LIN {X 0,Y 231.927,Z 556.531,A -85,B 0,C 180,E1 4341.378,E2 4341.378} C_VEL
LIN {X 0,Y 242.397,Z 520.672,A -85,B 0,C 180,E1 4340.064,E2 4340.064} C_VEL
LIN {X 0,Y 252.164,Z 483.622,A -85,B 0,C 180,E1 4339.103,E2 4339.103} C_VEL
LIN {X 0,Y 261.218,Z 444.481,A -85,B 0,C 180,E1 4338.33,E2 4338.33} C_VEL
LIN {X 0,Y 260.42,Z 444.342,A -85,B 0,C 180,E1 4336.736,E2 4336.736} C_VEL
LIN {X 0,Y 258.559,Z 446.515,A -85,B 0,C 180,E1 4332.054,E2 4332.054} C_VEL
LIN {X 0,Y 257.976,Z 449.054,A -85,B 0,C 180,E1 4329.369,E2 4329.369} C_VEL
LIN {X 0,Y 257.53,Z 454.171,A -85,B 0,C 180,E1 4325.906,E2 4325.906} C_VEL
LIN {X 0,Y 257.459,Z 455.233,A -85,B 0,C 180,E1 4325.433,E2 4325.433} C_VEL
LIN {X 0,Y 252.095,Z 484.028,A -85,B 0,C 180,E1 4321.933,E2 4321.933} C_VEL
LIN {X 0,Y 247.629,Z 509.442,A -85,B 0,C 180,E1 4318.236,E2 4318.236} C_VEL
LIN {X 0,Y 247.271,Z 511.086,A -85,B 0,C 180,E1 4318.085,E2 4318.085} C_VEL
LIN {X 0,Y 235.981,Z 546.89,A -85,B 0,C 180,E1 4317.26,E2 4317.26} C_VEL
LIN {X 0,Y 225.42,Z 575.954,A -85,B 0,C 180,E1 4316.366,E2 4316.366} C_VEL
LIN {X 0,Y 217.613,Z 594.168,A -85,B 0,C 180,E1 4315.587,E2 4315.587} C_VEL
LIN {X 0,Y 208.409,Z 612.205,A -85,B 0,C 180,E1 4314.557,E2 4314.557} C_VEL
LIN {X 0,Y 198.008,Z 629.617,A -85,B 0,C 180,E1 4313.241,E2 4313.241} C_VEL
LIN {X 0,Y 186.017,Z 646.929,A -85,B 0,C 180,E1 4311.498,E2 4311.498} C_VEL
LIN {X 0,Y 172.734,Z 663.594,A -85,B 0,C 180,E1 4309.228,E2 4309.228} C_VEL
LIN {X 0,Y 168.365,Z 668.643,A -85,B 0,C 180,E1 4308.388,E2 4308.388} C_VEL
LIN {X 0,Y 163.029,Z 674.093,A -85,B 0,C 180,E1 4307.699,E2 4307.699} C_VEL
LIN {X 0,Y 147.644,Z 686.875,A -85,B 0,C 180,E1 4306.83,E2 4306.83} C_VEL
LIN {X 0,Y 142.043,Z 691.517,A -85,B 0,C 180,E1 4305.902,E2 4305.902} C_VEL
LIN {X 0,Y 126.649,Z 704.484,A -85,B 0,C 180,E1 4301.326,E2 4301.326} C_VEL
LIN {X 0,Y 111.309,Z 715.997,A -85,B 0,C 180,E1 4295.127,E2 4295.127} C_VEL
LIN {X 0,Y 97.462,Z 725.548,A -85,B 0,C 180,E1 4287.065,E2 4287.065} C_VEL
LIN {X 0,Y 85.648,Z 733.443,A -85,B 0,C 180,E1 4276.367,E2 4276.367} C_VEL
LIN {X 0,Y 76.93,Z 739.822,A -85,B 0,C 180,E1 4262.199,E2 4262.199} C_VEL
LIN {X 0,Y 73.123,Z 744.052,A -85,B 0,C 180,E1 4246.842,E2 4246.842} C_VEL
LIN {X 0,Y 73.014,Z 746.243,A -85,B 0,C 180,E1 4233.925,E2 4233.925} C_VEL
LIN {X 0,Y 73.05,Z 746.869,A -85,B 0,C 180,E1 4227.602,E2 4227.602} C_VEL
LIN {X 0,Y 72.811,Z 747.091,A -85,B 0,C 180,E1 4215.688,E2 4215.688} C_VEL
LIN {X 0,Y 76.296,Z 746.032,A -85,B 0,C 180,E1 4199.262,E2 4199.262} C_VEL
LIN {X 0,Y 85.813,Z 743.101,A -85,B 0,C 180,E1 4183.745,E2 4183.745} C_VEL
LIN {X 0,Y 100.024,Z 738.311,A -85,B 0,C 180,E1 4171.821,E2 4171.821} C_VEL
LIN {X 0,Y 101.886,Z 737.625,A -85,B 0,C 180,E1 4170.519,E2 4170.519} C_VEL
LIN {X 0,Y 89.481,Z 735.216,A -85,B 0,C 180,E1 4147.058,E2 4147.058} C_VEL
LIN {X 0,Y 98.204,Z 732.294,A -85,B 0,C 180,E1 4117.553,E2 4117.553} C_VEL
LIN {X 0,Y 85.177,Z 735.025,A -85,B 0,C 180,E1 4105.258,E2 4105.258} C_VEL
LIN {X 0,Y 76.898,Z 735.979,A -85,B 0,C 180,E1 4090.552,E2 4090.552} C_VEL
LIN {X 0,Y 73.529,Z 735.548,A -85,B 0,C 180,E1 4075.796,E2 4075.796} C_VEL
LIN {X 0,Y 73.059,Z 734.257,A -85,B 0,C 180,E1 4063.455,E2 4063.455} C_VEL
LIN {X 0,Y 74.498,Z 732.026,A -85,B 0,C 180,E1 4050.001,E2 4050.001} C_VEL
LIN {X 0,Y 79.613,Z 728.071,A -85,B 0,C 180,E1 4035.454,E2 4035.454} C_VEL
LIN {X 0,Y 88.821,Z 722.314,A -85,B 0,C 180,E1 4022.515,E2 4022.515} C_VEL
LIN {X 0,Y 101.148,Z 714.793,A -85,B 0,C 180,E1 4012.203,E2 4012.203} C_VEL
LIN {X 0,Y 115.684,Z 705.33,A -85,B 0,C 180,E1 4004.163,E2 4004.163} C_VEL
LIN {X 0,Y 130.96,Z 694.255,A -85,B 0,C 180,E1 3998.152,E2 3998.152} C_VEL
LIN {X 0,Y 145.553,Z 682.354,A -85,B 0,C 180,E1 3993.779,E2 3993.779} C_VEL
LIN {X 0,Y 159.873,Z 669.114,A -85,B 0,C 180,E1 3990.339,E2 3990.339} C_VEL
LIN {X 0,Y 173.705,Z 654.497,A -85,B 0,C 180,E1 3987.572,E2 3987.572} C_VEL
LIN {X 0,Y 186.472,Z 639.018,A -85,B 0,C 180,E1 3985.38,E2 3985.38} C_VEL
LIN {X 0,Y 198.513,Z 622.1,A -85,B 0,C 180,E1 3983.554,E2 3983.554} C_VEL
LIN {X 0,Y 208.854,Z 605.18,A -85,B 0,C 180,E1 3982.127,E2 3982.127} C_VEL
LIN {X 0,Y 218.344,Z 586.768,A -85,B 0,C 180,E1 3980.906,E2 3980.906} C_VEL
LIN {X 0,Y 226.49,Z 567.593,A -85,B 0,C 180,E1 3979.898,E2 3979.898} C_VEL
LIN {X 0,Y 233.499,Z 546.938,A -85,B 0,C 180,E1 3979.045,E2 3979.045} C_VEL
LIN {X 0,Y 244.93,Z 507.349,A -85,B 0,C 180,E1 3977.816,E2 3977.816} C_VEL
LIN {X 0,Y 255.69,Z 465.177,A -85,B 0,C 180,E1 3976.969,E2 3976.969} C_VEL
LIN {X 0,Y 258.645,Z 452.199,A -85,B 0,C 180,E1 3976.719,E2 3976.719} C_VEL
LIN {X 0,Y 256.749,Z 454.341,A -85,B 0,C 180,E1 3972.187,E2 3972.187} C_VEL
LIN {X 0,Y 256.151,Z 456.887,A -85,B 0,C 180,E1 3969.55,E2 3969.55} C_VEL
LIN {X 0,Y 255.599,Z 461.227,A -85,B 0,C 180,E1 3966.726,E2 3966.726} C_VEL
LIN {X 0,Y 249.853,Z 489.15,A -85,B 0,C 180,E1 3963.299,E2 3963.299} C_VEL
LIN {X 0,Y 245.184,Z 513.039,A -85,B 0,C 180,E1 3959.874,E2 3959.874} C_VEL
LIN {X 0,Y 233.743,Z 548.774,A -85,B 0,C 180,E1 3959.127,E2 3959.127} C_VEL
LIN {X 0,Y 223.065,Z 577.863,A -85,B 0,C 180,E1 3958.304,E2 3958.304} C_VEL
LIN {X 0,Y 214.174,Z 597.67,A -85,B 0,C 180,E1 3957.491,E2 3957.491} C_VEL
LIN {X 0,Y 203.868,Z 616.732,A -85,B 0,C 180,E1 3956.421,E2 3956.421} C_VEL
LIN {X 0,Y 192.194,Z 634.969,A -85,B 0,C 180,E1 3955.033,E2 3955.033} C_VEL
LIN {X 0,Y 179.557,Z 651.97,A -85,B 0,C 180,E1 3953.286,E2 3953.286} C_VEL
LIN {X 0,Y 165.992,Z 667.856,A -85,B 0,C 180,E1 3951.061,E2 3951.061} C_VEL
LIN {X 0,Y 151.711,Z 682.536,A -85,B 0,C 180,E1 3948.212,E2 3948.212} C_VEL
LIN {X 0,Y 142.043,Z 691.517,A -85,B 0,C 180,E1 3945.902,E2 3945.902} C_VEL
LIN {X 0,Y 136.354,Z 696.167,A -85,B 0,C 180,E1 3944.862,E2 3944.862} C_VEL
LIN {X 0,Y 119.782,Z 706.857,A -85,B 0,C 180,E1 3943.026,E2 3943.026} C_VEL
LIN {X 0,Y 113.801,Z 710.716,A -85,B 0,C 180,E1 3941.496,E2 3941.496} C_VEL
LIN {X 0,Y 98.528,Z 720.99,A -85,B 0,C 180,E1 3934.575,E2 3934.575} C_VEL
LIN {X 0,Y 84.395,Z 729.788,A -85,B 0,C 180,E1 3924.83,E2 3924.83} C_VEL
LIN {X 0,Y 73.344,Z 736.665,A -85,B 0,C 180,E1 3911.91,E2 3911.91} C_VEL
LIN {X 0,Y 66.581,Z 741.753,A -85,B 0,C 180,E1 3895.713,E2 3895.713} C_VEL
LIN {X 0,Y 64.817,Z 744.776,A -85,B 0,C 180,E1 3879.768,E2 3879.768} C_VEL
LIN {X 0,Y 65.191,Z 745.925,A -85,B 0,C 180,E1 3869.999,E2 3869.999} C_VEL
LIN {X 0,Y 64.739,Z 746.384,A -85,B 0,C 180,E1 3860.217,E2 3860.217} C_VEL
LIN {X 0,Y 66.978,Z 745.975,A -85,B 0,C 180,E1 3842.432,E2 3842.432} C_VEL
LIN {X 0,Y 75.85,Z 743.765,A -85,B 0,C 180,E1 3824.614,E2 3824.614} C_VEL
LIN {X 0,Y 90.062,Z 739.719,A -85,B 0,C 180,E1 3811.256,E2 3811.256} C_VEL
LIN {X 0,Y 92.206,Z 739.054,A -85,B 0,C 180,E1 3809.829,E2 3809.829} C_VEL
LIN {X 0,Y 81.468,Z 736.055,A -85,B 0,C 180,E1 3778.591,E2 3778.591} C_VEL
LIN {X 0,Y 89.081,Z 734.092,A -85,B 0,C 180,E1 3758.402,E2 3758.402} C_VEL
LIN {X 0,Y 75.847,Z 736.262,A -85,B 0,C 180,E1 3744.82,E2 3744.82} C_VEL
LIN {X 0,Y 67.888,Z 736.673,A -85,B 0,C 180,E1 3728.214,E2 3728.214} C_VEL
LIN {X 0,Y 65.237,Z 735.79,A -85,B 0,C 180,E1 3712.531,E2 3712.531} C_VEL
LIN {X 0,Y 65.231,Z 734.421,A -85,B 0,C 180,E1 3699.708,E2 3699.708} C_VEL
LIN {X 0,Y 67.843,Z 731.656,A -85,B 0,C 180,E1 3684.08,E2 3684.08} C_VEL
LIN {X 0,Y 75.219,Z 727.026,A -85,B 0,C 180,E1 3668.15,E2 3668.15} C_VEL
LIN {X 0,Y 86.527,Z 720.71,A -85,B 0,C 180,E1 3655.514,E2 3655.514} C_VEL
LIN {X 0,Y 99.893,Z 713,A -85,B 0,C 180,E1 3646.32,E2 3646.32} C_VEL
LIN {X 0,Y 114.962,Z 703.477,A -85,B 0,C 180,E1 3639.281,E2 3639.281} C_VEL
LIN {X 0,Y 130.352,Z 692.534,A -85,B 0,C 180,E1 3634.065,E2 3634.065} C_VEL
LIN {X 0,Y 145.602,Z 680.199,A -85,B 0,C 180,E1 3630.089,E2 3630.089} C_VEL
LIN {X 0,Y 160.433,Z 666.472,A -85,B 0,C 180,E1 3626.975,E2 3626.975} C_VEL
LIN {X 0,Y 174.682,Z 651.299,A -85,B 0,C 180,E1 3624.482,E2 3624.482} C_VEL
LIN {X 0,Y 187.779,Z 635.16,A -85,B 0,C 180,E1 3622.509,E2 3622.509} C_VEL
LIN {X 0,Y 200.087,Z 617.461,A -85,B 0,C 180,E1 3620.859,E2 3620.859} C_VEL
LIN {X 0,Y 211.092,Z 598.668,A -85,B 0,C 180,E1 3619.511,E2 3619.511} C_VEL
LIN {X 0,Y 220.286,Z 579.718,A -85,B 0,C 180,E1 3618.445,E2 3618.445} C_VEL
LIN {X 0,Y 228.105,Z 559.864,A -85,B 0,C 180,E1 3617.567,E2 3617.567} C_VEL
LIN {X 0,Y 239.315,Z 523.749,A -85,B 0,C 180,E1 3616.37,E2 3616.37} C_VEL
LIN {X 0,Y 249.393,Z 487.249,A -85,B 0,C 180,E1 3615.539,E2 3615.539} C_VEL
LIN {X 0,Y 255.931,Z 460.666,A -85,B 0,C 180,E1 3615.059,E2 3615.059} C_VEL
LIN {X 0,Y 254.914,Z 462.238,A -85,B 0,C 180,E1 3612.229,E2 3612.229} C_VEL
LIN {X 0,Y 254.24,Z 464.93,A -85,B 0,C 180,E1 3609.622,E2 3609.622} C_VEL
LIN {X 0,Y 253.819,Z 467.409,A -85,B 0,C 180,E1 3608.025,E2 3608.025} C_VEL
LIN {X 0,Y 247.589,Z 495.193,A -85,B 0,C 180,E1 3604.561,E2 3604.561} C_VEL
LIN {X 0,Y 243.22,Z 515.223,A -85,B 0,C 180,E1 3601.684,E2 3601.684} C_VEL
LIN {X 0,Y 231.728,Z 550.784,A -85,B 0,C 180,E1 3601.025,E2 3601.025} C_VEL
LIN {X 0,Y 221.972,Z 577.219,A -85,B 0,C 180,E1 3600.358,E2 3600.358} C_VEL
LIN {X 0,Y 212.973,Z 596.994,A -85,B 0,C 180,E1 3599.633,E2 3599.633} C_VEL
LIN {X 0,Y 202.525,Z 615.982,A -85,B 0,C 180,E1 3598.672,E2 3598.672} C_VEL
LIN {X 0,Y 191.158,Z 633.557,A -85,B 0,C 180,E1 3597.473,E2 3597.473} C_VEL
LIN {X 0,Y 178.428,Z 650.486,A -85,B 0,C 180,E1 3595.912,E2 3595.912} C_VEL
LIN {X 0,Y 164.895,Z 666.126,A -85,B 0,C 180,E1 3593.948,E2 3593.948} C_VEL
LIN {X 0,Y 150.655,Z 680.543,A -85,B 0,C 180,E1 3591.442,E2 3591.442} C_VEL
LIN {X 0,Y 135.25,Z 694.226,A -85,B 0,C 180,E1 3588.055,E2 3588.055} C_VEL
LIN {X 0,Y 119.313,Z 706.716,A -85,B 0,C 180,E1 3583.447,E2 3583.447} C_VEL
LIN {X 0,Y 113.801,Z 710.716,A -85,B 0,C 180,E1 3581.496,E2 3581.496} C_VEL
LIN {X 0,Y 107.822,Z 714.499,A -85,B 0,C 180,E1 3579.766,E2 3579.766} C_VEL
LIN {X 0,Y 90.724,Z 722.93,A -85,B 0,C 180,E1 3575.995,E2 3575.995} C_VEL
LIN {X 0,Y 84.871,Z 725.894,A -85,B 0,C 180,E1 3573.333,E2 3573.333} C_VEL
LIN {X 0,Y 71.334,Z 733.478,A -85,B 0,C 180,E1 3561.712,E2 3561.712} C_VEL
LIN {X 0,Y 61.387,Z 739.358,A -85,B 0,C 180,E1 3545.478,E2 3545.478} C_VEL
LIN {X 0,Y 57.059,Z 743.284,A -85,B 0,C 180,E1 3526.281,E2 3526.281} C_VEL
LIN {X 0,Y 57.148,Z 745.006,A -85,B 0,C 180,E1 3512.004,E2 3512.004} C_VEL
LIN {X 0,Y 56.946,Z 745.501,A -85,B 0,C 180,E1 3504.962,E2 3504.962} C_VEL
LIN {X 0,Y 57.868,Z 745.639,A -85,B 0,C 180,E1 3486.582,E2 3486.582} C_VEL
LIN {X 0,Y 65.392,Z 744.248,A -85,B 0,C 180,E1 3466.521,E2 3466.521} C_VEL
LIN {X 0,Y 79.393,Z 741.014,A -85,B 0,C 180,E1 3451.085,E2 3451.085} C_VEL
LIN {X 0,Y 82.344,Z 740.172,A -85,B 0,C 180,E1 3448.659,E2 3448.659} C_VEL
LIN {X 0,Y 73.885,Z 737.24,A -85,B 0,C 180,E1 3416.118,E2 3416.118} C_VEL
LIN {X 0,Y 79.674,Z 735.688,A -85,B 0,C 180,E1 3399.246,E2 3399.246} C_VEL
LIN {X 0,Y 66.49,Z 737.23,A -85,B 0,C 180,E1 3384.298,E2 3384.298} C_VEL
LIN {X 0,Y 59.017,Z 737.12,A -85,B 0,C 180,E1 3365.583,E2 3365.583} C_VEL
LIN {X 0,Y 57.096,Z 736.046,A -85,B 0,C 180,E1 3348.969,E2 3348.969} C_VEL
LIN {X 0,Y 57.624,Z 734.434,A -85,B 0,C 180,E1 3334.979,E2 3334.979} C_VEL
LIN {X 0,Y 61.623,Z 731.454,A -85,B 0,C 180,E1 3317.825,E2 3317.825} C_VEL
LIN {X 0,Y 71,Z 726.46,A -85,B 0,C 180,E1 3301.394,E2 3301.394} C_VEL
LIN {X 0,Y 84.147,Z 719.739,A -85,B 0,C 180,E1 3289.193,E2 3289.193} C_VEL
LIN {X 0,Y 99.7,Z 711.143,A -85,B 0,C 180,E1 3280.345,E2 3280.345} C_VEL
LIN {X 0,Y 115.076,Z 701.614,A -85,B 0,C 180,E1 3274.369,E2 3274.369} C_VEL
LIN {X 0,Y 131.278,Z 690.135,A -85,B 0,C 180,E1 3269.744,E2 3269.744} C_VEL
LIN {X 0,Y 146.249,Z 678.015,A -85,B 0,C 180,E1 3266.414,E2 3266.414} C_VEL
LIN {X 0,Y 161.545,Z 663.76,A -85,B 0,C 180,E1 3263.649,E2 3263.649} C_VEL
LIN {X 0,Y 175.809,Z 648.336,A -85,B 0,C 180,E1 3261.484,E2 3261.484} C_VEL
LIN {X 0,Y 189.075,Z 631.638,A -85,B 0,C 180,E1 3259.731,E2 3259.731} C_VEL
LIN {X 0,Y 201.146,Z 613.797,A -85,B 0,C 180,E1 3258.301,E2 3258.301} C_VEL
LIN {X 0,Y 211.403,Z 595.847,A -85,B 0,C 180,E1 3257.18,E2 3257.18} C_VEL
LIN {X 0,Y 220.271,Z 577.219,A -85,B 0,C 180,E1 3256.252,E2 3256.252} C_VEL
LIN {X 0,Y 227.508,Z 558.613,A -85,B 0,C 180,E1 3255.515,E2 3255.515} C_VEL
LIN {X 0,Y 238.253,Z 524.713,A -85,B 0,C 180,E1 3254.479,E2 3254.479} C_VEL
LIN {X 0,Y 248.043,Z 490.171,A -85,B 0,C 180,E1 3253.751,E2 3253.751} C_VEL
LIN {X 0,Y 253.427,Z 469.215,A -85,B 0,C 180,E1 3253.409,E2 3253.409} C_VEL
LIN {X 0,Y 252.464,Z 471.884,A -85,B 0,C 180,E1 3250.497,E2 3250.497} C_VEL
LIN {X 0,Y 252.09,Z 473.738,A -85,B 0,C 180,E1 3249.316,E2 3249.316} C_VEL
LIN {X 0,Y 245.34,Z 501.367,A -85,B 0,C 180,E1 3245.816,E2 3245.816} C_VEL
LIN {X 0,Y 241.517,Z 517.381,A -85,B 0,C 180,E1 3243.523,E2 3243.523} C_VEL
LIN {X 0,Y 228.758,Z 556.164,A -85,B 0,C 180,E1 3242.89,E2 3242.89} C_VEL
LIN {X 0,Y 219.835,Z 579.4,A -85,B 0,C 180,E1 3242.347,E2 3242.347} C_VEL
LIN {X 0,Y 210.56,Z 599.032,A -85,B 0,C 180,E1 3241.684,E2 3241.684} C_VEL
LIN {X 0,Y 199.991,Z 617.668,A -85,B 0,C 180,E1 3240.819,E2 3240.819} C_VEL
LIN {X 0,Y 187.975,Z 635.633,A -85,B 0,C 180,E1 3239.684,E2 3239.684} C_VEL
LIN {X 0,Y 174.56,Z 652.795,A -85,B 0,C 180,E1 3238.199,E2 3238.199} C_VEL
LIN {X 0,Y 159.82,Z 669.041,A -85,B 0,C 180,E1 3236.241,E2 3236.241} C_VEL
LIN {X 0,Y 143.872,Z 684.258,A -85,B 0,C 180,E1 3233.613,E2 3233.613} C_VEL
LIN {X 0,Y 127.836,Z 697.52,A -85,B 0,C 180,E1 3230.228,E2 3230.228} C_VEL
LIN {X 0,Y 111.473,Z 709.38,A -85,B 0,C 180,E1 3225.625,E2 3225.625} C_VEL
LIN {X 0,Y 96.045,Z 719.312,A -85,B 0,C 180,E1 3219.54,E2 3219.54} C_VEL
LIN {X 0,Y 84.871,Z 725.894,A -85,B 0,C 180,E1 3213.333,E2 3213.333} C_VEL
LIN {X 0,Y 79.154,Z 728.768,A -85,B 0,C 180,E1 3210.256,E2 3210.256} C_VEL
LIN {X 0,Y 62.482,Z 734.88,A -85,B 0,C 180,E1 3201.549,E2 3201.549} C_VEL
LIN {X 0,Y 57.977,Z 736.722,A -85,B 0,C 180,E1 3196.45,E2 3196.45} C_VEL
LIN {X 0,Y 50.298,Z 741.362,A -85,B 0,C 180,E1 3175.932,E2 3175.932} C_VEL
LIN {X 0,Y 48.957,Z 743.971,A -85,B 0,C 180,E1 3155.859,E2 3155.859} C_VEL
LIN {X 0,Y 49.195,Z 744.496,A -85,B 0,C 180,E1 3148.834,E2 3148.834} C_VEL
LIN {X 0,Y 49.198,Z 745.046,A -85,B 0,C 180,E1 3131.022,E2 3131.022} C_VEL
LIN {X 0,Y 55.947,Z 744.265,A -85,B 0,C 180,E1 3107.223,E2 3107.223} C_VEL
LIN {X 0,Y 70.16,Z 741.643,A -85,B 0,C 180,E1 3089.618,E2 3089.618} C_VEL
LIN {X 0,Y 72.738,Z 741.051,A -85,B 0,C 180,E1 3087.474,E2 3087.474} C_VEL
LIN {X 0,Y 66.117,Z 738.349,A -85,B 0,C 180,E1 3054.791,E2 3054.791} C_VEL
LIN {X 0,Y 70.619,Z 737.081,A -85,B 0,C 180,E1 3040.648,E2 3040.648} C_VEL
LIN {X 0,Y 57.634,Z 738.062,A -85,B 0,C 180,E1 3024.627,E2 3024.627} C_VEL
LIN {X 0,Y 50.498,Z 737.577,A -85,B 0,C 180,E1 3003.672,E2 3003.672} C_VEL
LIN {X 0,Y 49.08,Z 736.345,A -85,B 0,C 180,E1 2986.573,E2 2986.573} C_VEL
LIN {X 0,Y 50.232,Z 734.568,A -85,B 0,C 180,E1 2970.002,E2 2970.002} C_VEL
LIN {X 0,Y 56.532,Z 730.935,A -85,B 0,C 180,E1 2949.627,E2 2949.627} C_VEL
LIN {X 0,Y 67.845,Z 725.705,A -85,B 0,C 180,E1 2933.88,E2 2933.88} C_VEL
LIN {X 0,Y 82.814,Z 718.584,A -85,B 0,C 180,E1 2922.568,E2 2922.568} C_VEL
LIN {X 0,Y 98.888,Z 710.034,A -85,B 0,C 180,E1 2915.017,E2 2915.017} C_VEL
LIN {X 0,Y 116.025,Z 699.566,A -85,B 0,C 180,E1 2909.498,E2 2909.498} C_VEL
LIN {X 0,Y 132.026,Z 688.239,A -85,B 0,C 180,E1 2905.684,E2 2905.684} C_VEL
LIN {X 0,Y 147.487,Z 675.624,A -85,B 0,C 180,E1 2902.783,E2 2902.783} C_VEL
LIN {X 0,Y 162.254,Z 661.727,A -85,B 0,C 180,E1 2900.502,E2 2900.502} C_VEL
LIN {X 0,Y 175.774,Z 647.047,A -85,B 0,C 180,E1 2898.72,E2 2898.72} C_VEL
LIN {X 0,Y 188.449,Z 631.13,A -85,B 0,C 180,E1 2897.249,E2 2897.249} C_VEL
LIN {X 0,Y 199.767,Z 614.576,A -85,B 0,C 180,E1 2896.059,E2 2896.059} C_VEL
LIN {X 0,Y 209.699,Z 597.528,A -85,B 0,C 180,E1 2895.087,E2 2895.087} C_VEL
LIN {X 0,Y 218.691,Z 579.134,A -85,B 0,C 180,E1 2894.242,E2 2894.242} C_VEL
LIN {X 0,Y 226.273,Z 560.145,A -85,B 0,C 180,E1 2893.545,E2 2893.545} C_VEL
LIN {X 0,Y 236.936,Z 527.466,A -85,B 0,C 180,E1 2892.615,E2 2892.615} C_VEL
LIN {X 0,Y 246.877,Z 493.326,A -85,B 0,C 180,E1 2891.949,E2 2891.949} C_VEL
LIN {X 0,Y 250.794,Z 478.527,A -85,B 0,C 180,E1 2891.732,E2 2891.732} C_VEL
LIN {X 0,Y 250.376,Z 480.034,A -85,B 0,C 180,E1 2890.615,E2 2890.615} C_VEL
LIN {X 0,Y 243.584,Z 505.96,A -85,B 0,C 180,E1 2887.311,E2 2887.311} C_VEL
LIN {X 0,Y 240.025,Z 519.579,A -85,B 0,C 180,E1 2885.386,E2 2885.386} C_VEL
LIN {X 0,Y 228.303,Z 555.116,A -85,B 0,C 180,E1 2884.904,E2 2884.904} C_VEL
LIN {X 0,Y 220.144,Z 576.604,A -85,B 0,C 180,E1 2884.492,E2 2884.492} C_VEL
LIN {X 0,Y 211.479,Z 595.284,A -85,B 0,C 180,E1 2883.979,E2 2883.979} C_VEL
LIN {X 0,Y 201.302,Z 613.582,A -85,B 0,C 180,E1 2883.286,E2 2883.286} C_VEL
LIN {X 0,Y 189.634,Z 631.344,A -85,B 0,C 180,E1 2882.368,E2 2882.368} C_VEL
LIN {X 0,Y 176.51,Z 648.429,A -85,B 0,C 180,E1 2881.161,E2 2881.161} C_VEL
LIN {X 0,Y 161.981,Z 664.704,A -85,B 0,C 180,E1 2879.564,E2 2879.564} C_VEL
LIN {X 0,Y 146.127,Z 680.035,A -85,B 0,C 180,E1 2877.416,E2 2877.416} C_VEL
LIN {X 0,Y 129.562,Z 693.868,A -85,B 0,C 180,E1 2874.571,E2 2874.571} C_VEL
LIN {X 0,Y 112.476,Z 706.238,A -85,B 0,C 180,E1 2870.654,E2 2870.654} C_VEL
LIN {X 0,Y 95.195,Z 717.128,A -85,B 0,C 180,E1 2865.08,E2 2865.08} C_VEL
LIN {X 0,Y 78.154,Z 726.512,A -85,B 0,C 180,E1 2856.637,E2 2856.637} C_VEL
LIN {X 0,Y 63.841,Z 733.75,A -85,B 0,C 180,E1 2844.526,E2 2844.526} C_VEL
LIN {X 0,Y 57.977,Z 736.722,A -85,B 0,C 180,E1 2836.45,E2 2836.45} C_VEL
LIN {X 0,Y 53.622,Z 738.588,A -85,B 0,C 180,E1 2830.103,E2 2830.103} C_VEL
LIN {X 0,Y 45.23,Z 741.066,A -85,B 0,C 180,E1 2817.357,E2 2817.357} C_VEL
LIN {X 0,Y 41.18,Z 742.489,A -85,B 0,C 180,E1 2804.371,E2 2804.371} C_VEL
LIN {X 0,Y 40.885,Z 742.917,A -85,B 0,C 180,E1 2799.737,E2 2799.737} C_VEL
LIN {X 0,Y 41.204,Z 743.743,A -85,B 0,C 180,E1 2788.607,E2 2788.607} C_VEL
LIN {X 0,Y 41.747,Z 744.34,A -85,B 0,C 180,E1 2765.971,E2 2765.971} C_VEL
LIN {X 0,Y 50.777,Z 743.557,A -85,B 0,C 180,E1 2739.827,E2 2739.827} C_VEL
LIN {X 0,Y 62.999,Z 741.68,A -85,B 0,C 180,E1 2725.901,E2 2725.901} C_VEL
LIN {X 0,Y 61.206,Z 738.346,A -85,B 0,C 180,E1 2682.099,E2 2682.099} C_VEL
LIN {X 0,Y 47.529,Z 738.736,A -85,B 0,C 180,E1 2662.401,E2 2662.401} C_VEL
LIN {X 0,Y 41.714,Z 737.73,A -85,B 0,C 180,E1 2638.648,E2 2638.648} C_VEL
LIN {X 0,Y 41.259,Z 736.394,A -85,B 0,C 180,E1 2619.769,E2 2619.769} C_VEL
LIN {X 0,Y 44.88,Z 733.778,A -85,B 0,C 180,E1 2597.129,E2 2597.129} C_VEL
LIN {X 0,Y 55.553,Z 729.206,A -85,B 0,C 180,E1 2576.088,E2 2576.088} C_VEL
LIN {X 0,Y 70.491,Z 722.953,A -85,B 0,C 180,E1 2562.476,E2 2562.476} C_VEL
LIN {X 0,Y 86.812,Z 715.289,A -85,B 0,C 180,E1 2553.979,E2 2553.979} C_VEL
LIN {X 0,Y 104.25,Z 705.804,A -85,B 0,C 180,E1 2548.072,E2 2548.072} C_VEL
LIN {X 0,Y 120.521,Z 695.503,A -85,B 0,C 180,E1 2544.137,E2 2544.137} C_VEL
LIN {X 0,Y 136.211,Z 684.028,A -85,B 0,C 180,E1 2541.214,E2 2541.214} C_VEL
LIN {X 0,Y 152.118,Z 670.56,A -85,B 0,C 180,E1 2538.828,E2 2538.828} C_VEL
LIN {X 0,Y 166.286,Z 656.682,A -85,B 0,C 180,E1 2537.052,E2 2537.052} C_VEL
LIN {X 0,Y 180.071,Z 641.071,A -85,B 0,C 180,E1 2535.556,E2 2535.556} C_VEL
LIN {X 0,Y 192.482,Z 624.692,A -85,B 0,C 180,E1 2534.354,E2 2534.354} C_VEL
LIN {X 0,Y 203.967,Z 606.884,A -85,B 0,C 180,E1 2533.331,E2 2533.331} C_VEL
LIN {X 0,Y 214.031,Z 588.263,A -85,B 0,C 180,E1 2532.486,E2 2532.486} C_VEL
LIN {X 0,Y 222.654,Z 568.838,A -85,B 0,C 180,E1 2531.776,E2 2531.776} C_VEL
LIN {X 0,Y 231.757,Z 542.999,A -85,B 0,C 180,E1 2531.041,E2 2531.041} C_VEL
LIN {X 0,Y 243.206,Z 506.178,A -85,B 0,C 180,E1 2530.27,E2 2530.27} C_VEL
LIN {X 0,Y 244.809,Z 500.666,A -85,B 0,C 180,E1 2530.167,E2 2530.167} C_VEL
LIN {X 0,Y 238.823,Z 521.809,A -85,B 0,C 180,E1 2527.27,E2 2527.27} C_VEL
LIN {X 0,Y 226.593,Z 558.532,A -85,B 0,C 180,E1 2526.868,E2 2526.868} C_VEL
LIN {X 0,Y 218.38,Z 579.409,A -85,B 0,C 180,E1 2526.519,E2 2526.519} C_VEL
LIN {X 0,Y 208.934,Z 598.845,A -85,B 0,C 180,E1 2526.044,E2 2526.044} C_VEL
LIN {X 0,Y 197.848,Z 617.797,A -85,B 0,C 180,E1 2525.395,E2 2525.395} C_VEL
LIN {X 0,Y 185.047,Z 636.201,A -85,B 0,C 180,E1 2524.516,E2 2524.516} C_VEL
LIN {X 0,Y 170.816,Z 653.543,A -85,B 0,C 180,E1 2523.357,E2 2523.357} C_VEL
LIN {X 0,Y 156.063,Z 669.023,A -85,B 0,C 180,E1 2521.901,E2 2521.901} C_VEL
LIN {X 0,Y 139.979,Z 683.591,A -85,B 0,C 180,E1 2519.933,E2 2519.933} C_VEL
LIN {X 0,Y 123.12,Z 696.773,A -85,B 0,C 180,E1 2517.282,E2 2517.282} C_VEL
LIN {X 0,Y 104.692,Z 709.16,A -85,B 0,C 180,E1 2513.334,E2 2513.334} C_VEL
LIN {X 0,Y 86.95,Z 719.402,A -85,B 0,C 180,E1 2507.8,E2 2507.8} C_VEL
LIN {X 0,Y 69.536,Z 728.124,A -85,B 0,C 180,E1 2499.167,E2 2499.167} C_VEL
LIN {X 0,Y 54.018,Z 735.163,A -85,B 0,C 180,E1 2484.989,E2 2484.989} C_VEL
LIN {X 0,Y 43.693,Z 740.142,A -85,B 0,C 180,E1 2463.31,E2 2463.31} C_VEL
LIN {X 0,Y 40.885,Z 742.917,A -85,B 0,C 180,E1 2439.737,E2 2439.737} C_VEL
LIN {X 0,Y 40.285,Z 743.487,A -85,B 0,C 180,E1 2432.123,E2 2432.123} C_VEL
LIN {X 0,Y 38.481,Z 743.834,A -85,B 0,C 180,E1 2421.97,E2 2421.97} C_VEL
LIN {X 0,Y 36.752,Z 743.598,A -85,B 0,C 180,E1 2391.762,E2 2391.762} C_VEL
LIN {X 0,Y 38.312,Z 743.494,A -85,B 0,C 180,E1 2386.018,E2 2386.018} C_VEL
LIN {X 0,Y 53.324,Z 742.04,A -85,B 0,C 180,E1 2363.771,E2 2363.771} C_VEL
LIN {X 0,Y 52.081,Z 739.325,A -85,B 0,C 180,E1 2324.405,E2 2324.405} C_VEL
LIN {X 0,Y 38.261,Z 739.161,A -85,B 0,C 180,E1 2301.631,E2 2301.631} C_VEL
LIN {X 0,Y 33.362,Z 737.971,A -85,B 0,C 180,E1 2274.811,E2 2274.811} C_VEL
LIN {X 0,Y 33.655,Z 736.528,A -85,B 0,C 180,E1 2253.409,E2 2253.409} C_VEL
LIN {X 0,Y 39.868,Z 733.582,A -85,B 0,C 180,E1 2226.345,E2 2226.345} C_VEL
LIN {X 0,Y 53.476,Z 728.631,A -85,B 0,C 180,E1 2206.229,E2 2206.229} C_VEL
LIN {X 0,Y 70.428,Z 721.95,A -85,B 0,C 180,E1 2194.574,E2 2194.574} C_VEL
LIN {X 0,Y 88.007,Z 713.86,A -85,B 0,C 180,E1 2187.606,E2 2187.606} C_VEL
LIN {X 0,Y 106.306,Z 703.881,A -85,B 0,C 180,E1 2182.82,E2 2182.82} C_VEL
LIN {X 0,Y 123.149,Z 693.097,A -85,B 0,C 180,E1 2179.644,E2 2179.644} C_VEL
LIN {X 0,Y 139.259,Z 681.096,A -85,B 0,C 180,E1 2177.271,E2 2177.271} C_VEL
LIN {X 0,Y 154.549,Z 667.891,A -85,B 0,C 180,E1 2175.431,E2 2175.431} C_VEL
LIN {X 0,Y 169.446,Z 652.921,A -85,B 0,C 180,E1 2173.912,E2 2173.912} C_VEL
LIN {X 0,Y 182.955,Z 637.123,A -85,B 0,C 180,E1 2172.708,E2 2172.708} C_VEL
LIN {X 0,Y 195.045,Z 620.649,A -85,B 0,C 180,E1 2171.729,E2 2171.729} C_VEL
LIN {X 0,Y 206.183,Z 602.759,A -85,B 0,C 180,E1 2170.89,E2 2170.89} C_VEL
LIN {X 0,Y 216.355,Z 583.097,A -85,B 0,C 180,E1 2170.151,E2 2170.151} C_VEL
LIN {X 0,Y 224.586,Z 563.495,A -85,B 0,C 180,E1 2169.56,E2 2169.56} C_VEL
LIN {X 0,Y 232.017,Z 542.264,A -85,B 0,C 180,E1 2169.033,E2 2169.033} C_VEL
LIN {X 0,Y 222.059,Z 570.144,A -85,B 0,C 180,E1 2168.761,E2 2168.761} C_VEL
LIN {X 0,Y 212.764,Z 590.675,A -85,B 0,C 180,E1 2168.423,E2 2168.423} C_VEL
LIN {X 0,Y 202.426,Z 609.479,A -85,B 0,C 180,E1 2167.972,E2 2167.972} C_VEL
LIN {X 0,Y 191.059,Z 626.941,A -85,B 0,C 180,E1 2167.39,E2 2167.39} C_VEL
LIN {X 0,Y 177.645,Z 644.442,A -85,B 0,C 180,E1 2166.581,E2 2166.581} C_VEL
LIN {X 0,Y 163.751,Z 660.037,A -85,B 0,C 180,E1 2165.579,E2 2165.579} C_VEL
LIN {X 0,Y 148.381,Z 674.926,A -85,B 0,C 180,E1 2164.225,E2 2164.225} C_VEL
LIN {X 0,Y 132.098,Z 688.54,A -85,B 0,C 180,E1 2162.424,E2 2162.424} C_VEL
LIN {X 0,Y 114.982,Z 700.872,A -85,B 0,C 180,E1 2159.958,E2 2159.958} C_VEL
LIN {X 0,Y 97.172,Z 711.882,A -85,B 0,C 180,E1 2156.44,E2 2156.44} C_VEL
LIN {X 0,Y 78.94,Z 721.5,A -85,B 0,C 180,E1 2151.092,E2 2151.092} C_VEL
LIN {X 0,Y 60.877,Z 729.637,A -85,B 0,C 180,E1 2142.285,E2 2142.285} C_VEL
LIN {X 0,Y 44.513,Z 736.168,A -85,B 0,C 180,E1 2126.209,E2 2126.209} C_VEL
LIN {X 0,Y 34.488,Z 740.559,A -85,B 0,C 180,E1 2099.526,E2 2099.526} C_VEL
LIN {X 0,Y 33.187,Z 742.828,A -85,B 0,C 180,E1 2071.724,E2 2071.724} C_VEL
LIN {X 0,Y 32.901,Z 743.247,A -85,B 0,C 180,E1 2061.257,E2 2061.257} C_VEL
LIN {X 0,Y 37.52,Z 743.523,A -85,B 0,C 180,E1 2028.22,E2 2028.22} C_VEL
LIN {X 0,Y 38.312,Z 743.494,A -85,B 0,C 180,E1 2026.018,E2 2026.018} C_VEL
LIN {X 0,Y 40.436,Z 743.27,A -85,B 0,C 180,E1 2018.667,E2 2018.667} C_VEL
LIN {X 0,Y 41.855,Z 742.801,A -85,B 0,C 180,E1 2010.107,E2 2010.107} C_VEL
LIN {X 0,Y 42.528,Z 742.227,A -85,B 0,C 180,E1 2001.518,E2 2001.518} C_VEL
LIN {X 0,Y 42.433,Z 741.723,A -85,B 0,C 180,E1 1994.039,E2 1994.039} C_VEL
LIN {X 0,Y 42.242,Z 741.59,A -85,B 0,C 180,E1 1991.907,E2 1991.907} C_VEL
LIN {X 0,Y 42.989,Z 740.15,A -85,B 0,C 180,E1 1967.663,E2 1967.663} C_VEL
LIN {X 0,Y 28.783,Z 739.449,A -85,B 0,C 180,E1 1939.844,E2 1939.844} C_VEL
LIN {X 0,Y 25.191,Z 738.211,A -85,B 0,C 180,E1 1910.933,E2 1910.933} C_VEL
LIN {X 0,Y 26.624,Z 736.65,A -85,B 0,C 180,E1 1883.535,E2 1883.535} C_VEL
LIN {X 0,Y 36.556,Z 733.203,A -85,B 0,C 180,E1 1853.009,E2 1853.009} C_VEL
LIN {X 0,Y 53.05,Z 727.865,A -85,B 0,C 180,E1 1835.864,E2 1835.864} C_VEL
LIN {X 0,Y 71.675,Z 720.781,A -85,B 0,C 180,E1 1826.776,E2 1826.776} C_VEL
LIN {X 0,Y 90.24,Z 712.262,A -85,B 0,C 180,E1 1821.455,E2 1821.455} C_VEL
LIN {X 0,Y 108.259,Z 702.381,A -85,B 0,C 180,E1 1817.959,E2 1817.959} C_VEL
LIN {X 0,Y 126.495,Z 690.534,A -85,B 0,C 180,E1 1815.352,E2 1815.352} C_VEL
LIN {X 0,Y 143.905,Z 677.188,A -85,B 0,C 180,E1 1813.414,E2 1813.414} C_VEL
LIN {X 0,Y 160.421,Z 662.219,A -85,B 0,C 180,E1 1811.895,E2 1811.895} C_VEL
LIN {X 0,Y 175.041,Z 646.722,A -85,B 0,C 180,E1 1810.741,E2 1810.741} C_VEL
LIN {X 0,Y 188.714,Z 629.703,A -85,B 0,C 180,E1 1809.777,E2 1809.777} C_VEL
LIN {X 0,Y 189.271,Z 628.94,A -85,B 0,C 180,E1 1809.733,E2 1809.733} C_VEL
LIN {X 0,Y 175.163,Z 646.757,A -85,B 0,C 180,E1 1809.066,E2 1809.066} C_VEL
LIN {X 0,Y 160.112,Z 662.964,A -85,B 0,C 180,E1 1808.197,E2 1808.197} C_VEL
LIN {X 0,Y 144.067,Z 677.787,A -85,B 0,C 180,E1 1807.046,E2 1807.046} C_VEL
LIN {X 0,Y 126.528,Z 691.674,A -85,B 0,C 180,E1 1805.443,E2 1805.443} C_VEL
LIN {X 0,Y 108.091,Z 704.104,A -85,B 0,C 180,E1 1803.183,E2 1803.183} C_VEL
LIN {X 0,Y 88.986,Z 714.952,A -85,B 0,C 180,E1 1799.842,E2 1799.842} C_VEL
LIN {X 0,Y 70.279,Z 723.876,A -85,B 0,C 180,E1 1794.788,E2 1794.788} C_VEL
LIN {X 0,Y 51.557,Z 731.343,A -85,B 0,C 180,E1 1785.845,E2 1785.845} C_VEL
LIN {X 0,Y 35.192,Z 736.982,A -85,B 0,C 180,E1 1768.464,E2 1768.464} C_VEL
LIN {X 0,Y 25.668,Z 740.73,A -85,B 0,C 180,E1 1735.367,E2 1735.367} C_VEL
LIN {X 0,Y 25.26,Z 742.156,A -85,B 0,C 180,E1 1709.996,E2 1709.996} C_VEL
LIN {X 0,Y 27.21,Z 742.853,A -85,B 0,C 180,E1 1673.928,E2 1673.928} C_VEL
LIN {X 0,Y 41.325,Z 742.305,A -85,B 0,C 180,E1 1643.154,E2 1643.154} C_VEL
LIN {X 0,Y 43.799,Z 742.134,A -85,B 0,C 180,E1 1640.609,E2 1640.609} C_VEL
LIN {X 0,Y 42.242,Z 741.59,A -85,B 0,C 180,E1 1631.907,E2 1631.907} C_VEL
LIN {X 0,Y 40.87,Z 741.293,A -85,B 0,C 180,E1 1626.419,E2 1626.419} C_VEL
LIN {X 0,Y 37.813,Z 741.032,A -85,B 0,C 180,E1 1619.951,E2 1619.951} C_VEL
LIN {X 0,Y 33.137,Z 740.804,A -85,B 0,C 180,E1 1612.23,E2 1612.23} C_VEL
LIN {X 0,Y 25.393,Z 740.346,A -85,B 0,C 180,E1 1598.335,E2 1598.335} C_VEL
LIN {X 0,Y 19.171,Z 739.568,A -85,B 0,C 180,E1 1575.906,E2 1575.906} C_VEL
LIN {X 0,Y 17.506,Z 738.049,A -85,B 0,C 180,E1 1533.28,E2 1533.28} C_VEL
LIN {X 0,Y 25.956,Z 735.342,A -85,B 0,C 180,E1 1491.954,E2 1491.954} C_VEL
LIN {X 0,Y 42.479,Z 730.829,A -85,B 0,C 180,E1 1472.078,E2 1472.078} C_VEL
LIN {X 0,Y 62.069,Z 724.367,A -85,B 0,C 180,E1 1462.747,E2 1462.747} C_VEL
LIN {X 0,Y 81.865,Z 716.239,A -85,B 0,C 180,E1 1457.704,E2 1457.704} C_VEL
LIN {X 0,Y 101.217,Z 706.488,A -85,B 0,C 180,E1 1454.519,E2 1454.519} C_VEL
LIN {X 0,Y 119.745,Z 695.267,A -85,B 0,C 180,E1 1452.332,E2 1452.332} C_VEL
LIN {X 0,Y 137.372,Z 682.624,A -85,B 0,C 180,E1 1450.708,E2 1450.708} C_VEL
LIN {X 0,Y 143.253,Z 677.962,A -85,B 0,C 180,E1 1450.223,E2 1450.223} C_VEL
LIN {X 0,Y 125.547,Z 691.671,A -85,B 0,C 180,E1 1449.059,E2 1449.059} C_VEL
LIN {X 0,Y 106.877,Z 703.925,A -85,B 0,C 180,E1 1447.411,E2 1447.411} C_VEL
LIN {X 0,Y 88.335,Z 714.211,A -85,B 0,C 180,E1 1445.096,E2 1445.096} C_VEL
LIN {X 0,Y 69.01,Z 723.147,A -85,B 0,C 180,E1 1441.406,E2 1441.406} C_VEL
LIN {X 0,Y 49.203,Z 730.628,A -85,B 0,C 180,E1 1434.688,E2 1434.688} C_VEL
LIN {X 0,Y 30.802,Z 736.282,A -85,B 0,C 180,E1 1420.273,E2 1420.273} C_VEL
LIN {X 0,Y 18.227,Z 740.047,A -85,B 0,C 180,E1 1383.263,E2 1383.263} C_VEL
LIN {X 0,Y 17.164,Z 741.423,A -85,B 0,C 180,E1 1348.326,E2 1348.326} C_VEL
LIN {X 0,Y 23.052,Z 742.175,A -85,B 0,C 180,E1 1294.493,E2 1294.493} C_VEL
LIN {X 0,Y 34.501,Z 741.89,A -85,B 0,C 180,E1 1275.113,E2 1275.113} C_VEL
LIN {X 0,Y 34.01,Z 740.813,A -85,B 0,C 180,E1 1252.626,E2 1252.626} C_VEL
LIN {X 0,Y 19.559,Z 739.639,A -85,B 0,C 180,E1 1218.338,E2 1218.338} C_VEL
LIN {X 0,Y 19.171,Z 739.568,A -85,B 0,C 180,E1 1215.906,E2 1215.906} C_VEL
LIN {X 0,Y 16.523,Z 738.939,A -85,B 0,C 180,E1 1196.355,E2 1196.355} C_VEL
LIN {X 0,Y 14.711,Z 738.004,A -85,B 0,C 180,E1 1161.736,E2 1161.736} C_VEL
LIN {X 0,Y 21.571,Z 735.952,A -85,B 0,C 180,E1 1116.782,E2 1116.782} C_VEL
LIN {X 0,Y 25.389,Z 735.084,A -85,B 0,C 180,E1 1111.117,E2 1111.117} C_VEL
LIN {X 0,Y 44.607,Z 730.169,A -85,B 0,C 180,E1 1099.713,E2 1099.713} C_VEL
LIN {X 0,Y 65.072,Z 723.363,A -85,B 0,C 180,E1 1094.533,E2 1094.533} C_VEL
LIN {X 0,Y 85.715,Z 714.672,A -85,B 0,C 180,E1 1091.526,E2 1091.526} C_VEL
LIN {X 0,Y 92.608,Z 711.336,A -85,B 0,C 180,E1 1090.739,E2 1090.739} C_VEL
LIN {X 0,Y 72.66,Z 720.762,A -85,B 0,C 180,E1 1088.709,E2 1088.709} C_VEL
LIN {X 0,Y 52.206,Z 728.579,A -85,B 0,C 180,E1 1085.2,E2 1085.2} C_VEL
LIN {X 0,Y 31.032,Z 734.883,A -85,B 0,C 180,E1 1077.157,E2 1077.157} C_VEL
LIN {X 0,Y 12.397,Z 739.186,A -85,B 0,C 180,E1 1045.646,E2 1045.646} C_VEL
LIN {X 0,Y 9.096,Z 740.654,A -85,B 0,C 180,E1 986.836,E2 986.836} C_VEL
LIN {X 0,Y 19.604,Z 741.436,A -85,B 0,C 180,E1 914.277,E2 914.277} C_VEL
LIN {X 0,Y 25.707,Z 741.41,A -85,B 0,C 180,E1 906.693,E2 906.693} C_VEL
LIN {X 0,Y 25.603,Z 741.208,A -85,B 0,C 180,E1 901.367,E2 901.367} C_VEL
LIN {X 0,Y 11.177,Z 739.838,A -85,B 0,C 180,E1 863.638,E2 863.638} C_VEL
LIN {X 0,Y 10.227,Z 738.434,A -85,B 0,C 180,E1 797.96,E2 797.96} C_VEL
LIN {X 0,Y 22.903,Z 735.671,A -85,B 0,C 180,E1 753.963,E2 753.963} C_VEL
LIN {X 0,Y 25.389,Z 735.084,A -85,B 0,C 180,E1 751.117,E2 751.117} C_VEL
LIN {X 0,Y 25.205,Z 735.127,A -85,B 0,C 180,E1 748.992,E2 748.992} C_VEL
LIN {X 0,Y 22.289,Z 735.816,A -85,B 0,C 180,E1 744.709,E2 744.709} C_VEL
LIN {X 0,Y 16.163,Z 737.109,A -85,B 0,C 180,E1 739.486,E2 739.486} C_VEL
LIN {X 0,Y 7.21,Z 738.757,A -85,B 0,C 180,E1 727.323,E2 727.323} C_VEL
LIN {X 0,Y 2.546,Z 739.461,A -85,B 0,C 180,E1 707.951,E2 707.951} C_VEL
LIN {X 0,Y 1.341,Z 739.909,A -85,B 0,C 180,E1 581.693,E2 581.693} C_VEL
LIN {X 0,Y 4.31,Z 740.11,A -85,B 0,C 180,E1 542.156,E2 542.156} C_VEL
LIN {X 0,Y 6.561,Z 738.72,A -85,B 0,C 180,E1 383.915,E2 383.915} C_VEL
LIN {X 0,Y 24.587,Z 735.515,A -85,B 0,C 180,E1 372.596,E2 372.596} C_VEL
LIN {X 0,Y 27.576,Z 734.888,A -85,B 0,C 180,E1 371.787,E2 371.787} C_VEL
LIN {X 0,Y 8.026,Z 738.68,A -85,B 0,C 180,E1 364.833,E2 364.833} C_VEL
LIN {X 0,Y 2.546,Z 739.461,A -85,B 0,C 180,E1 347.951,E2 347.951} C_VEL
LIN {X 0,Y 1.185,Z 741.442,A -85,B 0,C 180,E1 312.301,E2 312.301} C_VEL
LIN {X 0,Y 1.185,Z 786.5,A -85,B 0,C 180,E1 312.301,E2 312.301} C_VEL
LIN {X 0,Y 1.185,Z 786.5,A -85,B 0,C 180,E1 312.301,E2 312.301}

QRS_NEXT_CUT()

QRS_NEXT()
QRS_HOME()

END
